# B&R Automation Studio project AAU12Segmenter (part 4)

### Config_1.assembly6d - X20CP1685/mapp6D/Config_1.assembly6d
```
Element gAssembly6D_1 (Type=assembly6d)
  Simulation6D = SimOff
  Shuttles:
    MaxShuttleCount = 8
    ShuttleIDMode = RealTimeID
    DefaultPosition:
      DefZ = 1.0
      DefRx = 0
      DefRy = 0
      DefRz = 0
    Limits:
      InPlaneLimits:
        InPlaneVelLim = 2
        InPlaneAccLim = 10
        InPlaneEmergDec = 1
      ShortAxLim:
        ShortAxAccLim:
          AccZLim = 10.0
          AccRxLim = 10.0
          AccRyLim = 10.0
          AccRzLim = 10.0
        ShortAxVelLim:
          VelZLim = 0.15
          VelRxLim = 0.1
          VelRyLim = 0.1
          VelRzLim = 0.3
  CyclicChannel6D:
    ReadChannel:
      Xaxis = TRUE
      Yaxis = TRUE
      Zaxis = TRUE
      Rxaxis = TRUE
      Ryaxis = TRUE
      Rzaxis = TRUE
  Fieldbus6D:
    SyncMode6D = ExternalPlkSync
    NodeNumber = 20
  IOMapp:
    Input = ::FBin
    Output = ::FBout
  Layout:
    Layout6D[1] = Layout6D_1
```

### Config_2.layout6d - X20CP1685/mapp6D/Config_2.layout6d
```
Element Layout6D_1 (Type=layout6d)
  Segments:
    SegRow = 4
    SegCol = 3
    Segment[1]:
      X = 0
      Y = 0
      Name
      IsMaster = True
    Segment[2]:
      X = 0
      Y = 1
      Name
      IsMaster = False
    Segment[3]:
      X = 0
      Y = 2
      Name
      IsMaster = False
    Segment[4]:
      X = 0
      Y = 3
      Name
      IsMaster = False
    Segment[5]:
      X = 1
      Y = 0
      Name
      IsMaster = False
    Segment[6]:
      X = 1
      Y = 1
      Name
      IsMaster = False
    Segment[7]:
      X = 1
      Y = 2
      Name
      IsMaster = False
    Segment[8]:
      X = 1
      Y = 3
      Name
      IsMaster = False
    Segment[9]:
      X = 2
      Y = 0
      Name
      IsMaster = False
    Segment[10]:
      X = 2
      Y = 1
      Name
      IsMaster = False
    Segment[11]:
      X = 2
      Y = 2
      Name
      IsMaster = False
    Segment[12]:
      X = 2
      Y = 3
      Name
      IsMaster = False
```

## Logical view

Binary libraries used (declarations not repeated): operator, runtime, astime, AsIecCon, standard, brdkSTR, AsSem, sys_lib, brsystem, AsBrStr, AsZip, FileIO, AsARCfg, AsEPL, AsIO, IecCheck, brdkViBase, brdkViCal, brdkViGeom, brdkViImg, brdkViMapp, brdkViVF, BRSE_RTK, AsHttp, powerlnk, MTLinAlg, ViBase 5.19.1, CoTrace 5.19.0, McBase, SfDomain 5.19.0, MpBase 5.19.0, McAcp6D, KUKAmxA3_1 3.01.1, AsUDP, asstring, KUKAmxA3_2 3.02.0, KUKAmxA3_3 3.03.1, KUKAmxA3_0 3.00.2

### Global.var - Global variables
```iecst
VAR
	FBin : Mc6DControllerFBIOType;
	FBout : Mc6DControllerFBIOType;
	GripperBlackPin : BOOL;
END_VAR
```

### Package Logical/Libraries - Global libraries

### Library Logical/Libraries/brdkMU (ANSIC) - BRDK machine unit library. Provides functionality to control machines.

#### brdkCM.typ
```iecst
TYPE
	brdk_cm_setup_typ : 	STRUCT  (*Equipment module setup structure.*)
		name : STRING[BRDK_MU_NAME_STRING_SIZE]; (*Name of the module.*)
		nameIdx : DINT := -1; (*Index to be added to name. If -1 no index will be set.*)
		parent : brdk_mu_setup_module_typ; (*Parameters to setup a parent module.*)
		sibling : ARRAY[0..BRDK_MU_MAX_SIBLINGS]OF brdk_mu_setup_module_typ; (*Enables the logging of the last state and sub state.*)
		status : brdk_cm_setup_status_typ; (*Enables the logging of the last state and sub state.*)
	END_STRUCT;
	brdk_cm_setup_status_typ : 	STRUCT  (*Enable or disable status functionality.*)
		state : BOOL := TRUE; (*State string.*)
		last : BOOL := TRUE; (*Last log entries.*)
	END_STRUCT;
	brdk_cm_status_typ : 	STRUCT  (*Control module status type.*)
		ready : BOOL := FALSE; (*Control module is ready for use.*)
		state : STRING[BRDK_MU_MAX_DESCRIPTION_STRING]; (*Can be set in the task to descripe what the module is doing in this state.*)
		time : UDINT; (*[ms] Actual time spend in the current state.*)
		last : ARRAY[0..BRDK_MU_MAX_LAST_SIZE]OF STRING[25]; (*The last state the module was in.*)
		cycleTime : UDINT; (*[µsec] Cycle time of the modules's task.*)
		parent : brdk_mu_status_module_typ; (*Information about the parent.*)
		sibling : ARRAY[0..BRDK_MU_MAX_SIBLINGS]OF brdk_mu_status_module_typ; (*List of available siblings.*)
		sleeping : BOOL; (*Indicates that the module is sleeping meaning that the module is not being executed because a new instance is being transferred.*)
		level : UDINT; (*Level in the hierarchy. Parent is level 0.*)
		name : STRING[BRDK_MU_NAME_STRING_SIZE]; (*Name of the module.*)
	END_STRUCT;
	brdk_cm_internal_mu_list_typ : 	STRUCT  (*Holds index's in the MU list.*)
		idx : DINT := -1; (*Own index in the mu list.*)
		parentIdx : DINT := -1; (*Parent index in the mu list.*)
		siblingIdx : ARRAY[0..BRDK_MU_MAX_SIBLINGS]OF DINT := [4(-1)]; (*Siblings index in the mu list.*)
	END_STRUCT;
	brdk_cm_internal_typ : 	STRUCT  (*Control module internal variables.*)
		initSubstate : UINT := 0; (*Internal temp sub state to be used in INIT PROGRAM.*)
		muList : brdk_cm_internal_mu_list_typ; (*Holds index's in the MU list.*)
		old : brdk_cm_state_old_typ; (*Holds the old states.*)
	END_STRUCT;
	brdk_cm_state_old_typ : 	STRUCT  (*Holds the old states.*)
		state : UINT; (*Old CM state.*)
		substate : UINT; (*Old CM substate.*)
	END_STRUCT;
END_TYPE
```

#### brdkEM.typ
```iecst
TYPE
	brdk_em_states_typ :
		( (*Module states. Based on ISA–TR88.00.02 state model.*)
		STATE_DEACTIVATED := 0, (*State Type: Wait
The module has not been activated yet. An activate command will cause an exit from
DEACTIVATED to a ACTIVATING state.*)
		STATE_CLEARING := 1, (*State Type: Acting
Initiated by a state command to clear faults that may have occurred
when ABORTING, and are present in the ABORTED state before
proceeding to a STOPPED state.*)
		STATE_STOPPED := 2, (*State Type: Wait
The machine is powered and stationary after completing the
STOPPING state. All communications with other systems are
functioning (if applicable). A Reset command will cause an exit from
STOPPED to the RESETTING state.*)
		STATE_STARTING := 3, (*State Type: Acting
This state provides the steps needed to start the machine and is a
result of a starting type command (local or remote). Following this
command the machine will begin to Execute.*)
		STATE_IDLE := 4, (*State Type: Wait
This is a state which indicates that RESETTING is complete. This
state maintains the machine conditions which were achieved during
the RESETTING state, and performs operations required when the
machine is in IDLE.*)
		STATE_SUSPENDED := 5, (*State Type: Wait
The machine may be running at a relevant set point speed, but
there is no product being produced while the machine is waiting for
external process conditions to return to normal. When the offending
process conditions return to normal, the SUSPENDED state will
transition to UNSUSPENDING and hence continue towards the
normal EXECUTE state.*)
		STATE_EXECUTE := 6, (*State Type: Dual
Once the machine is processing materials it is deemed to be
executing or in the EXECUTE state. Different machine modes will
result in specific types of EXECUTE activities. For example, if the
machine is in the Production mode, the EXECUTE will result in
products being produced, while in Clean Out mode the EXECUTE
state refers to the action of cleaning the machine.*)
		STATE_STOPPING := 7, (*State Type: Acting
This state executes the logic which brings the machine to a
controlled stop as reflected by the STOPPED state. Normal
STARTING of the machine can not be initiated unless RESETTING
had taken place.*)
		STATE_ABORTING := 8, (*State Type: Acting
The ABORTED state can be entered at any time in response to the
Abort command or on the occurrence of a machine fault. The
aborting logic will bring the machine to a rapid safe stop. Operation
of the emergency stop will cause the machine to be tripped by its
safety system. It will also provide a signal to initiate the
ABORTING State.*)
		STATE_ABORTED := 9, (*State Type: Wait
This state maintains machine status information relevant to the
Abort condition. The machine can only exit the ABORTED state
after an explicit Clear command, subsequently to manual
intervention to correct and reset the detected machine faults.*)
		STATE_HOLDING := 10, (*State Type: Acting
When the machine is in the EXECUTE state, the Hold command
can be used to start HOLDING logic which brings the machine to a
controlled stop or to a state which represents HELD for the
particular unit control mode. A machine can go into this state either
when an internal equipment fault is automatically detected or by an
operator command. The Hold command offers the operator a safe
way to intervene manually in the process (such as removing a
broken bottle from the in-feed) and restarting execution when
conditions are safe. To be able to restart production correctly after
the HELD state, all relevant process set-points and return status of
the procedures at the time of receiving the Hold command must be
saved in the machine controller when executing the HOLDING
procedure.*)
		STATE_HELD := 11, (*State Type: Wait
The HELD state holds the machine's operation while material
blockages are cleared, or to stop throughput while a downstream
problem is resolved, or enable the safe correction of an equipment
fault before the production may be resumed.*)
		STATE_UNHOLDING := 12, (*State Type: Acting
The UNHOLDING state is a response to an Operator command to
resume the EXECUTE state. Issuing the Unhold command will
retrieve the saved set-points and return the status conditions to
prepare the machine to re-enter the normal EXECUTE state.*)
		STATE_SUSPENDING := 13, (*State Type: Acting
This state is a result of a change in monitored conditions due to
process conditions or factors. The trigger event will cause a
temporary suspension of the EXECUTE state. SUSPENDING is
typically the result of starvation of upstream material in-feeds (i.e.,
container feed, beverage feed, crown feed, lubricant feed, etc.) that
is outside the dynamic speed control range or a downstream outfeed
blockage that prevents the machine from EXECUTING
continued steady production. During the controlled sequence of
SUSPENDING the machine will transition to a SUSPENDED state.
The SUSPENDING state might be forced by the operator.*)
		STATE_UNSUSPENDING := 14, (*State Type: Acting
This state is a result of a machine generated request from
SUSPENDED state to go back to the EXECUTE state. The actions
of this state may include ramping up speeds, turning on vacuums,
and the re-engagement of clutches. This state is done prior to
EXECUTE state, and prepares the machine for the EXECUTE state.*)
		STATE_RESETTING := 15, (*State Type: Acting
This state is the result of a RESET command from the STOPPED or
complete state. RESETTING will typically cause a machine to
sound a horn and place the machine in a state where components
are energized awaiting a START command.*)
		STATE_COMPLETING := 16, (*State Type: Acting
This state is an automatic response from the EXECUTE state.
Normal operation has run to completion (i.e., processing of material
at the infeed will stop).*)
		STATE_COMPLETE := 17, (*State Type: Wait
The machine has finished the COMPLETING state and is now
waiting for a Reset command before transitioning to the
RESETTING state.*)
		STATE_DEACTIVATING := 18, (*State Type: Acting
This state is the result of a disabled ACTIVATE command.*)
		STATE_ACTIVATING := 19 (*State Type: Acting
State between DEACTIVATED and STOPPED. This state is done prior to
STOPPED state, and prepares the machine for the STOPPED state.*)
		) := STATE_DEACTIVATED;
	brdk_em_activation_typ :
		( (*Type of activation of equipment module.*)
		BRDK_EM_ACTIVATE := 0, (*Activates the equipment module.*)
		BRDK_EM_DEACTIVATE := 1, (*Deactivated the equipment module.*)
		BRDK_EM_ACTIVATE_BY_PARENT := 2 (*Automatically follows it's parent activation.*)
		) := BRDK_EM_DEACTIVATE;
	brdk_em_command_typ : 	STRUCT  (*Equipment module commands. Based on ISATR88.00.02.*)
		abort : BOOL := FALSE; (*Abort --> Go to STATE_ABORTING - Can be set in all states.*)
		clear : BOOL := FALSE; (*Clear --> Go to STATE_STOPPING - Can only be set in STATE_ABORTED.*)
		stop : BOOL := FALSE; (*Stop --> Go to STATE_STOPPING - Can be set in all states.*)
		reset : BOOL := FALSE; (*Reset --> Go to STATE_RESETTING - Can only be set in STATE_STOPPED.*)
		start : BOOL := FALSE; (*Start --> Go to STATE_STARTING - Can only be set in STATE_IDLE, STATE_SUSPENDED, STATE_HELD.*)
		hold : BOOL := FALSE; (*Hold --> Go to STATE_HOLDING - Can only be set in STATE_EXECUTE.*)
		suspend : BOOL := FALSE; (*Suspend --> Go to STATE_SUSPENDING - Can only be set in STATE_EXECUTE.*)
		complete : BOOL := FALSE; (*Complete --> Go to STATE_COMPLETING - Can only be set in STATE_EXECUTE.*)
		sc : BOOL := FALSE; (*The State Complete indication within the Acting state procedure will cause a state transition to occur. Same functionality as subsuate = SC.*)
	END_STRUCT;
	brdk_em_setup_typ : 	STRUCT  (*Equipment module setup structure.*)
		name : STRING[BRDK_MU_NAME_STRING_SIZE]; (*Name of the module. If empty the name of the task will be given.*)
		nameIdx : DINT := -1; (*Index to be added to name. If -1 no index will be set.*)
		reactTo : brdk_em_setup_react_typ := BRDK_EM_REACT_TO_ALL; (*Indicates which parent state the module should react to.*)
		parent : brdk_mu_setup_module_typ; (*Parameters to setup a parent module.*)
		skipStopSC : BOOL := FALSE; (*When this parameter is set the module will stop even though is not in sub state SC.*)
		sibling : ARRAY[0..BRDK_MU_MAX_SIBLINGS]OF brdk_mu_setup_module_typ; (*List of siblings to a module.*)
		activation : brdk_em_activation_typ := BRDK_EM_ACTIVATE; (*Type of activation of equipment module.*)
		useSubstateSC : BOOL := FALSE; (*Enables the if substate is set to SC it will work as cmd.sc.*)
		restore : brdk_em_setup_restore_typ; (*Functionality to restore a module to it's state after a e.g. power failure.*)
		status : brdk_em_setup_status_typ; (*Enable or disable status functionality.*)
		customModeNames : ARRAY[0..BRDK_EM_MAX_CUSTOM_MODES]OF brdk_em_setup_custom_modes_typ; (*Custom mode names.*)
	END_STRUCT;
	brdk_em_setup_custom_modes_typ : 	STRUCT  (*Custom mode names.*)
		mode : DINT := 0; (*Mode integer value.*)
		modeName : STRING[BRDK_EM_MAX_MODE_NAME_SIZE] := ''; (*Mode name.*)
	END_STRUCT;
	brdk_em_setup_status_typ : 	STRUCT  (*Enable or disable status functionality.*)
		stateSubstateMode : BOOL := TRUE; (*State, sub state and mode strings.*)
		last : BOOL := TRUE; (*Last log entries.*)
		waitingFor : BOOL := TRUE; (*Waiting for.*)
		interruptedBy : BOOL := TRUE; (*interrupted by.*)
	END_STRUCT;
	brdk_em_setup_react_typ :
		( (*Indicates witch command/state the module should react to.*)
		BRDK_EM_REACT_TO_ALL := 0, (*Reacts to all states.*)
		BRDK_EM_REACT_TO_ABORT_AND_STOP := 1, (*Reacts only to abort and stop states.*)
		BRDK_EM_REACT_TO_ABORT_ONLY := 2, (*Reacts only to abort state.*)
		BRDK_EM_REACT_TO_STOP_ONLY := 3, (*Reacts only to stop state.*)
		BRDK_EM_REACT_TO_NONE := 4, (*Doesn't react to any state or mode change. Runs total independent. Equal to the old cmd.ignore.*)
		BRDK_EM_LISTEN_TO_ABORT_AND_STOP := 5, (*The module listen to it's parent aborting and stopping only. Parent don't react to the module.*)
		BRDK_EM_LISTEN_TO_ABORT_ONLY := 6, (*The module listen to it's parent aborting only. Parent don't react to the module.*)
		BRDK_EM_LISTEN_TO_STOP_ONLY := 7 (*The module listen to it's parent stopping only. Parent don't react to the module.*)
		) := BRDK_EM_REACT_TO_ALL;
	brdk_em_setup_restore_typ : 	STRUCT  (*Functionality to restore a module to it's state after a e.g. power failure.*)
		pRestoreStruct : REFERENCE TO brdk_em_restore_module_typ; (*Pointer to the restore structure. Must be defined directly in the task in order to make it retain/permanent.*)
		activate : BOOL := FALSE; (*Activates the storing of the module information in the restore structure. This is to avoid overwriting the restore information.*)
	END_STRUCT;
	brdk_em_status_typ : 	STRUCT  (*Equipment module status.*)
		state : STRING[21]; (*String representation of the state.*)
		substate : STRING[BRDK_MU_MAX_DESCRIPTION_STRING]; (*Can be set in the task to descripe what the module is doing in this substate.*)
		mode : STRING[21]; (*String representation of the mode.*)
		name : STRING[BRDK_MU_NAME_STRING_SIZE]; (*Name of the module. If empty the name of the task will be given.*)
		time : UDINT; (*[ms] Actual time spend in the current state.*)
		last : ARRAY[0..BRDK_MU_MAX_LAST_SIZE]OF STRING[43]; (*The last state and substate the module was in and the spend time.*)
		childCount : UDINT; (*How many children are registered.*)
		waitingFor : brdk_em_waiting_for_typ; (*Info: Which child the parent and the underlying modules are waiting for.*)
		interruptedBy : brdk_em_interrupted_by_typ; (*Info: Which child interruped the parent by going into STOPPING or ABORTING.*)
		color : brdk_em_color_typ; (*Color depending af the unit state.*)
		lightTree : brdk_em_status_light_tree_typ; (*Light tree indicating the status of the module.*)
		cycleTime : UDINT; (*[µsec] Cycle time of the modules's task.*)
		parent : brdk_mu_status_module_typ; (*Information about the parent.*)
		sibling : ARRAY[0..BRDK_MU_MAX_SIBLINGS]OF brdk_mu_status_module_typ; (*List of available siblings.*)
		unvalidatedCmd : BOOL; (*Indicates that the current state cannot accept the given command.*)
		unvalidatedMode : BOOL; (*Indicates that the current state cannot accept the given mode change. Modes can only be changed in STATE_STOPPED and in STATE_ACTIVATING. The status flag will be reset by a state change.*)
		sleeping : BOOL; (*Indicates that the module is sleeping meaning that the module is not being executed because a new instance is being transferred.*)
		level : UDINT; (*Level in the hierarchy. Parent is level 0.*)
	END_STRUCT;
	brdk_em_status_light_tree_typ : 	STRUCT  (*Light tree indicating the status of the module. The idea of the light tree status is that it can be mapped directly to an output module.*)
		red : BOOL := FALSE; (*Color red.*)
		yellow : BOOL := FALSE; (*Color yellow.*)
		blue : BOOL := FALSE; (*Color blue.*)
		green : BOOL := FALSE; (*Color green.*)
	END_STRUCT;
	brdk_em_color_typ :
		( (*Color to display the current state.*)
		GREY := 0, (*Wait State - Unit is disabled*)
		BLUE := 1, (*Wait State – A stable state used to identify that a Unit has achieved a defined set of
conditions. In such a state the Unit is holding or maintaining a status until transitioning
to an Acting state (White color). The unit is powered and stationary.*)
		WHITE := 2, (*Acting State – A state which represents some processing activity, for example ramping
up speed.
It implies the single or repeated execution of processing steps in a logical order, for a
finite time or until a specific condition has been reached, for example within the
Starting state the quality of the received data is checking, before raping up speed for
execution.*)
		GREEN := 3, (*Dual State - The Unit is in a stable acting state. The unit is running and drives are active
and the unit is producing.*)
		RED := 4, (*Wait state – A state which represents an error state on the Unit. In this state the Unit is
not producing, until the operator have managed to make a transition to the EXECUTING
state. The state holds the units operation in a safe environment, until the command
unhold are executed. For example a material blockage will move the unit into the HELD
state. The unit will leave the state HELD, when the operator have entered the unit,
removed the the bloackage, and enabled all safeguards and activated the Unhold
command.*)
		ORANGE := 5 (*Wait State – A state which represents an error state on the line and the Unit is running
at a relevant set point speed, but there is no product being produced while the unit is
waiting for external process conditions to return to normal. The unit will also enter this
state if the operator want to have a break.*)
		) := GREY;
	brdk_em_interrupted_by_typ : 	STRUCT  (*Tells which unit has interrupted the hierarchy into STATE_ABORTING or STATE_STOPPING.*)
		name : STRING[BRDK_MU_NAME_STRING_SIZE]; (*Name of the child that has interrupted the parent.*)
		state : brdk_em_states_typ := STATE_DEACTIVATED; (*State info.*)
		substate : UINT := 0; (*Substate info.*)
	END_STRUCT;
	brdk_em_waiting_for_typ : 	STRUCT  (*Tells which child module the hierarchy are waiting for. Can be that the modules are waiting for more children, but only one of them a shown at a time.*)
		name : STRING[BRDK_MU_NAME_STRING_SIZE]; (*Name of the child that the parent is waiting for.*)
		substate : STRING[BRDK_MU_MAX_DESCRIPTION_STRING]; (*Child substate.*)
	END_STRUCT;
	brdk_em_internal_typ : 	STRUCT  (*Internal variables.*)
		SemCreate_0 : SemCreate; (*Module semaphore.*)
		old : brdk_em_state_old_typ; (*Last state info.*)
		flashTime : UDINT := 0; (*Flash time counter.*)
		initSubstate : UINT := 0; (*Internal temp sub state to be used in STATE_DEACTIVATED.*)
		pInterrupter : UDINT := 0; (*Pointer to the module that interrupted.*)
		findParent : BOOL := FALSE; (*The module automatically finds it's parent's state.*)
		muList : brdk_em_internal_mu_list_typ; (*Holds index's in the MU list.*)
		cmdSC : BOOL; (*Internal command state complete.*)
		statusCnt : brdk_em_internal_status_cnt_typ; (*Status counter to indicate if a status change has been made.*)
		waitingForIdx : DINT := -1; (*Index of the module we are waiting for.*)
		deactivateRequest : BOOL := TRUE; (*A request to deactivate the mdule has been made.*)
		timeReminder : UDINT; (*Reminder of time when cycle time is below 1ms.*)
	END_STRUCT;
	brdk_em_internal_status_cnt_typ : 	STRUCT  (*Status counter to indicate if a status change has been made.*)
		internalCounter : DINT := -1; (*Internal counter which will be incremented if the status changes.*)
		externalCounter : DINT := -1; (*External counter which will hold the status counter of the waiting for module.*)
	END_STRUCT;
	brdk_em_state_old_typ : 	STRUCT  (*Holds the old states.*)
		state : brdk_em_states_typ := STATE_DEACTIVATED; (*Old state.*)
		substate : UINT := 0; (*Old substate.*)
		mode : DINT := 0; (*Old mode.*)
		reactTo : brdk_em_setup_react_typ := BRDK_EM_REACT_TO_ALL; (*Old reactTo.*)
	END_STRUCT;
	brdk_em_internal_mu_list_typ : 	STRUCT  (*Holds index's in the MU list.*)
		idx : DINT := -1; (*Own index in the mu list.*)
		parentIdx : DINT := -1; (*Parent index in the mu list.*)
		siblingIdx : ARRAY[0..BRDK_MU_MAX_SIBLINGS]OF DINT := [4(-1)]; (*Siblings index in the mu list.*)
		childrenIdx : ARRAY[0..BRDK_EM_MAX_CHILDREN]OF DINT; (*Children index in the mu list.*)
	END_STRUCT;
	brdk_em_restore_module_typ : 	STRUCT  (*Hold information that can be used to restore to it's active state in the case of a power failure.*)
		state : brdk_em_states_typ; (*Restored state.*)
		substate : UINT; (*Restored sub state.*)
		sc : BOOL; (*Restores state complete.*)
		mode : UINT; (*Restore mode.*)
	END_STRUCT;
	brdk_em_static_status_text_typ :
		( (*Internal enum to set a static status text*)
		STATUS_TEXT_DESCRIPTION := 0,
		STATUS_TEXT_ACTIVATION := 1
		);
END_TYPE
```

#### brdkMU.typ
```iecst
TYPE
	brdk_mu_setup_module_typ : 	STRUCT  (*Parameters to setup a connection to a module.*)
		name : STRING[BRDK_MU_NAME_STRING_SIZE]; (*Logical name of the module.*)
		index : DINT := -1; (*Index to be added to the module name. If -1 no index will be set.*)
	END_STRUCT;
	brdk_mu_status_module_typ : 	STRUCT  (*Status of a module.*)
		state : brdk_em_states_typ := STATE_DEACTIVATED; (*Module states. Based on ISA-TR88.00.02 state model.*)
		substate : UINT := 0; (*Equipment module substate can be used in the task. When a state is done set cmd.sc = true and the fb will take the unit to it's next state.*)
		sleeping : BOOL := FALSE; (*Indicates that the module is sleeping meaning that the module is not being executed because a new instance is being transferred.*)
		mode : DINT; (*Mode of the module.*)
		sc : BOOL; (*The State Complete indication within the Acting state procedure will cause a state transition to occur.*)
	END_STRUCT;
END_TYPE
```

#### brdkMU.fun
```iecst
FUNCTION_BLOCK brdkEM (*Represents an equipment module.*) (*$GROUP=User*)
	VAR_INPUT
		description : STRING[BRDK_MU_MAX_DESCRIPTION_STRING]; (*Description of what the substate is doing or waiting for.*)
		mode : DINT := MODE_PRODUCING; (*Control modes. Based on ISA-TR88.00.02 control modes. Modes can only be changed in STATE_STOPPED.*)
		cmd : brdk_em_command_typ; (*Control commands. Based on ISA-TR88.00.02 commands.*)
		setup : brdk_em_setup_typ; (*Setup of module.*)
		substate : UINT := 0; (*Equipment module substate can be used in the task. When a state is done set cmd.sc = true and the fb will take the unit to it's next state.*)
	END_VAR
	VAR_OUTPUT
		state : brdk_em_states_typ := STATE_DEACTIVATED; (*Equipment module state. State changes are controlled in the fb and is not allowed outside this fb. Based on ISA-TR88.00.02 states.*)
		status : brdk_em_status_typ; (*Module status.*)
	END_VAR
	VAR
		internal : brdk_em_internal_typ; (*Internal variables.*)
	END_VAR
END_FUNCTION_BLOCK

FUNCTION brdkEMSleep : DINT (*Put an equipment module to sleep. $RETURN=index;Index in the list.*) (*$GROUP=User,$CAT=User,$GROUPICON=User.png,$CATICON=User.png*)
	VAR_INPUT
		pEM : UDINT; (*Pointer to the equipment module.*)
	END_VAR
END_FUNCTION

FUNCTION brdkEMModeToA : UDINT (*Converts an equipment module mode int to a string representation. $RETURN=pointer;String pointer to mode string.*) (*$GROUP=User,$CAT=User,$GROUPICON=User.png,$CATICON=User.png*)
	VAR_INPUT
		mode : DINT := 0; (*Equipment module mode.*)
		pEM : UDINT := 0; (*Pointer to equipment module.*)
	END_VAR
END_FUNCTION

FUNCTION brdkEMStateToA : UDINT (*Converts an equipment module state enum to a string representation. $RETURN=pointer;String pointer to state string.*) (*$GROUP=User,$CAT=User,$GROUPICON=User.png,$CATICON=User.png*)
	VAR_INPUT
		state : brdk_em_states_typ; (*Equipment module state.*)
	END_VAR
END_FUNCTION

FUNCTION_BLOCK brdkCM (*Represents a control module. The module does not follow the ISA-TR88.00.02 standard.*) (*$GROUP=User,$CAT=User,$GROUPICON=User.png,$CATICON=User.png*)
	VAR_INPUT
		description : STRING[BRDK_MU_MAX_DESCRIPTION_STRING]; (*Description of what the state / substate is doing or waiting for.*)
		state : UINT := 0; (*Control module state must be used in the task.*)
		substate : UINT := 0; (*Control module substate must be used in the task.*)
		setup : brdk_cm_setup_typ; (*Setup of module.*)
	END_VAR
	VAR_OUTPUT
		status : brdk_cm_status_typ; (*Module status.*)
	END_VAR
	VAR
		internal : brdk_cm_internal_typ; (*Internal variables.*)
	END_VAR
END_FUNCTION_BLOCK

FUNCTION brdkCMSleep : DINT (*Put a control module to sleep. $RETURN=index;Index in the list.*) (*$GROUP=User,$CAT=User,$GROUPICON=User.png,$CATICON=User.png*)
	VAR_INPUT
		pCM : UDINT; (*Pointer to the control module.*)
	END_VAR
END_FUNCTION

FUNCTION brdkCMChangeParent : DINT (*Changes the parent of a control module. $RETURN=index;Index in the new parent.*) (*$GROUP=User,$CAT=User,$GROUPICON=User.png,$CATICON=User.png*)
	VAR_INPUT
		pCM : UDINT; (*Pointer to the control module.*)
		pParentName : UDINT; (*Pointert to the logical name of the parent module.*)
		parentIndex : DINT; (*Index to be added to the module name. If -1 no index will be set.*)
	END_VAR
END_FUNCTION

FUNCTION_BLOCK brdkUM (*Unit Machine / Information Receiver module. It makes communication with a remote system easy. This fb makes it possible to remote control an equipment module.*) (*$GROUP=User,$CAT=User,$GROUPICON=User.png,$CATICON=User.png*)
	VAR_INPUT
		mode : brdk_um_mode_typ := BRDK_UM_MODE_MANUAL; (*Communication mode.*)
		pEM : UDINT; (*Pointer to the main equipment module (machine unit).*)
		Status : brdk_um_pml_s_typ; (*Status tags.*)
		Admin : brdk_um_pml_a_typ; (*Administration tags.*)
	END_VAR
	VAR_OUTPUT
		Command : brdk_um_pml_c_typ; (*Command tags.*)
	END_VAR
	VAR
		internal : brdk_um_pml_internal_typ; (*Internal variables.*)
	END_VAR
END_FUNCTION_BLOCK
```

#### brdkMU_func.h
```c
#ifndef BRDK_MU_FUNCS
#define BRDK_MU_FUNCS 1

#include <brdkMU.h>
#include <bur/plctypes.h>

#ifdef __cplusplus
	extern "C"
	{
#endif

#ifdef __cplusplus
	};
#endif

#define false 0
#define true 1
#define NULL 0

extern SemCreate_typ SemCreateMUList;
extern unsigned char emListReady;

signed long addToMUList(unsigned long this, unsigned char type);
signed long getMUIndex(unsigned long this, brdk_mu_setup_module_typ* module);
brdkEM_typ* getEm(signed long idx);
signed long sleepMU(signed long idx, unsigned long this);
signed long wakeMU(signed long idx, unsigned long this);
unsigned long getCycleTime();
void updateSiblingInfo(signed long (*idxArr)[], brdk_mu_status_module_typ* status);
unsigned char moduleSleeping(signed long idx);

#endif /* !BRDK_MU_FUNCS */
```

#### brdkUM_func.h
```c
#ifndef BRDK_UM_FUNCS
#define BRDK_UM_FUNCS 1

#include <brdkMU_func.h>

void setCommand(signed long ctrlCmd, brdk_em_command_typ* emCmd, unsigned char value);
signed long cmdToState(signed long cmd);
void handleProductOverflow(brdk_um_pml_a_pc_typ* arr);

#endif /* !BRDK_UM_FUNCS */
```

#### brdkCM.c
```c
#include <brdkCM_func.h>

void brdkCM(struct brdkCM* this) {
	int i;
	brdkEM_typ* parent = getEm(this->internal.muList.parentIdx);
	brdk_mu_setup_module_typ module;

	/* initialize control module */
	switch(this->internal.initSubstate) {

		case 0:	/* this substate is only called in void _INIT / PROGRAM _INIT */
			if(this->setup.status.state) brdkStrCpy((unsigned long)this->status.state,(unsigned long)"initializing - looking for module pointers");
			if(this->setup.name[0] == 0) ST_name(0,(char*)&this->setup.name,(unsigned char)0); 														/* set module name to task name if not set*/
			brdkStrCpy((unsigned long)this->status.name,(unsigned long)this->setup.name);
			if(this->setup.nameIdx > -1) brdkStrAppendUdintToA(this->setup.nameIdx,(unsigned long)&this->status.name, BRDK_STR_CONVERT_DECIMAL,-1);	/* add index to task name */
			this->internal.muList.parentIdx = -1;
			for(i=0; i<= BRDK_MU_MAX_SIBLINGS; i++) this->internal.muList.siblingIdx[i] = -1;
			this->internal.initSubstate = 10;
			break;

		case 10:
			if(!emListReady) {
				if(this->setup.status.state) brdkStrCpy((unsigned long)this->status.state,(unsigned long)"waiting for mu list to be ready");
			}
			else {
				brdkStrCpy((unsigned long)module.name,(unsigned long)this->setup.name);
				module.index = this->setup.nameIdx;
				this->internal.muList.idx = getMUIndex((unsigned long)this, &module);
				if(this->internal.muList.idx != -1) {
					wakeMU(this->internal.muList.idx,(unsigned long)this);
					if(this->setup.status.last) {
						brdkStrMemMove((unsigned long)this->status.last[1],(unsigned long)this->status.last[0], sizeof(this->status.last[0])*BRDK_MU_MAX_LAST_SIZE);
						brdkStrCpy((unsigned long)this->status.last[0],(unsigned long)"module awake");
					}
					this->internal.initSubstate = 65001;
				}
				else {
					if(SemAcquire(SemCreateMUList.ident) != ERR_OK) {
						if(this->setup.status.state) brdkStrCpy((unsigned long)this->status.state,(unsigned long)"waiting global semaphore to be free");
					}
					else {
						this->internal.muList.idx = addToMUList((unsigned long)this,0);
						SemRelease(SemCreateMUList.ident);
						if(this->setup.status.state) brdkStrCpy((unsigned long)this->status.state,(unsigned long)"module added em list");
						if(this->internal.muList.idx != -1) this->internal.initSubstate = !this->setup.parent.name[0] ? 40 : 30;	/* check if the module has a parent name assigned */
						else {
							if(this->setup.status.state) brdkStrCpy((unsigned long)this->status.state,(unsigned long)"em list full. Expand BRDK_EM_MAX_EMS.");
							this->internal.initSubstate = 200;
						}
					}
				}
			}

		case 30:	/* find parent */
			this->internal.muList.parentIdx = getMUIndex((unsigned long)this, &this->setup.parent);
			if(this->internal.muList.parentIdx == -1) {
				if(this->setup.status.state) brdkStrCpy((unsigned long)this->status.state,(unsigned long)"parent not found");
			}
			else this->internal.initSubstate = 40;
			break;

		case 40:	/* find siblings */
			for(i=0; i<= BRDK_MU_MAX_SIBLINGS; i++) {
				if(this->setup.sibling[i].name[0] != 0) {
					this->internal.muList.siblingIdx[i] = getMUIndex((unsigned long)this, &this->setup.sibling[i]);
					if(this->internal.muList.siblingIdx[i] == -1) {
						if(this->setup.status.state) {
							brdkStrCpy((unsigned long)this->status.state,(unsigned long)"sibling: ");
							brdkStrCat((unsigned long)this->status.state,(unsigned long)this->setup.sibling[i].name);
							brdkStrCat((unsigned long)this->status.state,(unsigned long)" not found");
						}
						break;
					}
				}
			}
			if(i>=BRDK_MU_MAX_SIBLINGS) {
				this->status.state[0] = 0;	/* reset status text */
				this->internal.initSubstate = 65000;
			}
			break;

		case 65000:	/* module ready */
			/* check if status is not set */
			if(this->status.state[0] == 0 && this->setup.status.state) {
				brdkStrUdintToA(this->state,(unsigned long)this->status.state,BRDK_STR_CONVERT_DECIMAL);
				if(this->substate != 0) {
					brdkStrCat((unsigned long)this->status.state,(unsigned long)": ");
					brdkStrAppendUdintToA(this->substate,(unsigned long)this->status.state,BRDK_STR_CONVERT_DECIMAL,-1);
				}
				if(this->description[0] != 0) {
					brdkStrCat((unsigned long)this->status.state,(unsigned long)": ");
					brdkStrCat((unsigned long)this->status.state,(unsigned long)this->description);
				}
			}

			/* state change */
			if(this->state != this->internal.old.state || this->substate != this->internal.old.substate) {
				/* save last state for log */
				if(this->setup.status.last) {
					brdkStrMemMove((unsigned long)this->status.last[1],(unsigned long)this->status.last[0], sizeof(this->status.last[0])*BRDK_MU_MAX_LAST_SIZE);
					brdkStrUdintToA(this->internal.old.state,(unsigned long)this->status.last[0],BRDK_STR_CONVERT_DECIMAL);
					brdkStrCat((unsigned long)this->status.last[0],(unsigned long)": ");
					if(this->internal.old.substate || this->substate != 0) {	/* if the substate != 0 then we also want to log the oldsubstate even if it's 0 */
						brdkStrAppendUdintToA(this->internal.old.substate,(unsigned long)this->status.last[0],BRDK_STR_CONVERT_DECIMAL,-1);
						brdkStrCat((unsigned long)this->status.last[0], (unsigned long)": ");
					}
					brdkStrAppendUdintToA(this->status.time, (unsigned long)this->status.last[0],BRDK_STR_CONVERT_DECIMAL,-1);
					brdkStrCat((unsigned long)this->status.last[0], (unsigned long)"ms");
				}
				/* reset */
				if(this->state != this->internal.old.state) this->substate = 0;	/* if the state has been changed the substate will be reset */
				this->status.state[0] = this->description[0] = 0;
				this->internal.old.state = this->state;
				this->internal.old.substate = this->substate;
				this->status.time = 0;
			}
			else this->status.time += this->status.cycleTime/1000;

			/* update parent info */
			if(parent != NULL) {
				this->status.parent.state = parent->state;
				this->status.parent.substate = parent->substate;
				this->status.parent.sleeping = parent->status.sleeping;
				this->status.parent.sc = parent->cmd.sc;
			}

			/* update siblings info */
			updateSiblingInfo(&this->internal.muList.siblingIdx, &this->status.sibling[0]);

			this->status.level = parent != NULL ? parent->status.level+1 : 0;	/* sets the hierarchy level */

			break;

	}

	if(!this->status.cycleTime) this->status.cycleTime = getCycleTime();	/* get the modules cycle time */
	this->status.ready = this->internal.initSubstate == 65000;

}
```

#### brdkCMChangeParent.c
```c
#include <brdkMU_func.h>

signed long brdkCMChangeParent(unsigned long pCM, unsigned long pParentName, signed long parentIndex) {
	signed long tmpIdx = 0;
	brdk_mu_setup_module_typ module;
	brdkCM_typ* this;
	if(pCM != 0 && pParentName != 0 && emListReady) {
		this = (brdkCM_typ*)pCM;
		brdkStrCpy((unsigned long)module.name,pParentName);
		module.index = parentIndex;
		tmpIdx = getMUIndex((unsigned long)this, &module);
		if(tmpIdx != -1) {
			this->internal.muList.parentIdx = tmpIdx;
			brdkStrCpy((unsigned long)this->setup.parent.name,(unsigned long)module.name);
			this->setup.parent.index = module.index;
			return this->internal.muList.parentIdx;
		}
	}
	return -1;
}
```

#### brdkEM_func.c
```c
#include <brdkEM_func.h>

static unsigned char semCreator = false;
SemCreate_typ SemCreateMUList;
char tmpStr[BRDK_MU_MAX_DESCRIPTION_STRING];

/* initialize the equipment module */
void brdkEMInitialize(brdkEM_typ* this, brdkEM_typ* parent) {
	int i;
	brdk_mu_setup_module_typ module;

	switch(this->internal.initSubstate) {

		case 0:
			if(this->setup.name[0] == 0) ST_name(0,(char*)&this->setup.name,(unsigned char)0); 														/* set module name to task name if not set*/
			brdkStrCpy((unsigned long)this->status.name,(unsigned long)this->setup.name);
			if(this->setup.status.stateSubstateMode) {
				brdkStrCpy((unsigned long)this->status.state,(unsigned long)brdkEMStateToA(this->state));
				brdkStrCpy((unsigned long)this->status.mode,brdkEMModeToA(this->mode, this));
			}
			if(this->setup.nameIdx > -1) brdkStrAppendUdintToA(this->setup.nameIdx,(unsigned long)&this->status.name, BRDK_STR_CONVERT_DECIMAL,-1);	/* add index to task name */
			this->internal.muList.parentIdx = -1;
			for(i=0; i<= BRDK_EM_MAX_CHILDREN; i++) this->internal.muList.childrenIdx[i] = -1;
			for(i=0; i<= BRDK_MU_MAX_SIBLINGS; i++) this->internal.muList.siblingIdx[i] = -1;
			if(!semCreator) {
				setSubStateText(this,(unsigned long)"creating global semaphore");
				semCreator = true;
				this->internal.initSubstate = 10;
			}
			else this->internal.initSubstate = 20;
			break;

		case 10:
			SemCreateMUList.enable = true;
			SemCreateMUList.initCount = 0;
			SemCreateMUList.maxCount = 1;
			SemCreate(&SemCreateMUList);
			if(SemCreateMUList.status != ERR_OK) setSubStateText(this,(unsigned long)"creating global semaphore");
			else {
				SemRelease(SemCreateMUList.ident);
				this->internal.muList.idx = addToMUList((unsigned long)this,0);
				if(this->internal.muList.idx != -1) {
					emListReady = true;
					this->internal.initSubstate = !this->setup.parent.name[0] ? 40 : 30;	/* check if the module has a parent name assigned */
				}
				else {
					setSubStateText(this,(unsigned long)"em list full. Expand BRDK_EM_MAX_EMS.");
					this->internal.initSubstate = 200;
				}
			}
			break;

		case 20:	/* add module to em list */
			if(!emListReady) setSubStateText(this,(unsigned long)"waiting for em list to be ready");
			else {
				brdkStrCpy((unsigned long)module.name,(unsigned long)this->setup.name);
				module.index = this->setup.nameIdx;
				this->internal.muList.idx = getMUIndex((unsigned long)this, &module);
				if(this->internal.muList.idx != -1) {
					if(moduleSleeping(this->internal.muList.idx)) {
						wakeMU(this->internal.muList.idx,(unsigned long)this);
						if(this->setup.status.last) {
							brdkStrMemMove((unsigned long)this->status.last[1],(unsigned long)this->status.last[0], sizeof(this->status.last[0])*BRDK_MU_MAX_LAST_SIZE);
							brdkStrCpy((unsigned long)this->status.last[0],(unsigned long)"module awake");
						}
						this->internal.initSubstate = 65000;
					}
					else {	/* module name already exists in the list */
						this->status.substate[0] = 0;	/* reset sub state text */
						if(this->setup.status.stateSubstateMode) {
							brdkStrCpy((unsigned long)tmpStr,(unsigned long)"module name ");
							brdkStrCat((unsigned long)tmpStr,(unsigned long)module.name);
							brdkStrCat((unsigned long)tmpStr,(unsigned long)" already used. Rename module.");
							setSubStateText(this,(unsigned long)tmpStr);
						}
						this->internal.muList.idx = -1;
						this->internal.initSubstate = 100;
					}
				}
				else {
					if(SemAcquire(SemCreateMUList.ident) != ERR_OK) setSubStateText(this,(unsigned long)"waiting global semaphore to be free");
					else {
						this->internal.muList.idx = addToMUList((unsigned long)this,0);
						SemRelease(SemCreateMUList.ident);
						setSubStateText(this,(unsigned long)"module added em list");
						if(this->internal.muList.idx != -1) this->internal.initSubstate = !this->setup.parent.name[0] ? 40 : 30;	/* check if the module has a parent name assigned */
						else {
							setSubStateText(this,(unsigned long)"em list full. Expand BRDK_EM_MAX_EMS.");
							this->internal.initSubstate = 200;
						}
					}
				}
			}
			break;

		case 30:	/* find parent */
			this->internal.muList.parentIdx = getMUIndex((unsigned long)this, &this->setup.parent);
			if(this->internal.muList.parentIdx == -1) setSubStateText(this,(unsigned long)"parent not found");
			else this->internal.initSubstate = 40;
			break;

		case 40:	/* find siblings */
			for(i=0; i<= BRDK_MU_MAX_SIBLINGS; i++) {
				if(this->setup.sibling[i].name[0] != 0) {
					this->internal.muList.siblingIdx[i] = getMUIndex((unsigned long)this, &this->setup.sibling[i]);
					if(this->internal.muList.siblingIdx[i] == -1) {
						if(this->setup.status.stateSubstateMode) {
							brdkStrCpy((unsigned long)tmpStr,(unsigned long)"sibling: ");
							brdkStrCat((unsigned long)tmpStr,(unsigned long)this->setup.sibling[i].name);
							brdkStrCat((unsigned long)tmpStr,(unsigned long)" not found");
							setSubStateText(this,(unsigned long)tmpStr);
						}
						break;
					}
				}
			}
			if(i>=BRDK_MU_MAX_SIBLINGS) {
				this->status.substate[0] = 0;	/* reset status text */
				this->internal.initSubstate = this->internal.SemCreate_0.ident == 0 ? 50 : 60;
			}
			break;

		case 50:
			this->internal.SemCreate_0.enable = true;
			this->internal.SemCreate_0.initCount = 0;
			this->internal.SemCreate_0.maxCount = 1;
			SemCreate(&this->internal.SemCreate_0);
			switch(this->internal.SemCreate_0.status) {

				case 0:	/* ERR_OK */
					SemRelease(this->internal.SemCreate_0.ident);		/* release the semaphore so it's ready */
					this->internal.initSubstate = 60;
					break;

				case 65535:	/* ERR_FUB_BUSY */
					break;

				default:
					setSubStateText(this,(unsigned long)"error creating the semaphore");
					break;

			}
			break;

		case 60:
			switch(this->setup.activation) {
				case BRDK_EM_ACTIVATE:
					this->internal.deactivateRequest = false;
					this->internal.initSubstate = 70;
					break;

				case BRDK_EM_ACTIVATE_BY_PARENT:
					if(parent != NULL) {
						if(!parent->internal.deactivateRequest) {
							this->internal.initSubstate = 70;
							this->internal.deactivateRequest = false;
						}
					}
					break;

				default: break;

			}
			break;

		case 70:
			setSubStateText(this,(unsigned long)"register child to parent");
			if(RegisterChild(this, parent) == 0) {
				this->internal.initSubstate = 65000;				/* add child to parent's children list */
				if(this->substate == 0) this->substate = 65000;		/* if substate is still 0 it's auto set to SC */
			}
			break;

		case 100: /* error module name already used. Check if anme is being changed */
			break;

	}
}

/* traverse and find the real interrupter */
unsigned long findInterrupter(unsigned long pEM) {
	if(((brdkEM_typ*)pEM)->internal.pInterrupter != pEM) return findInterrupter(((brdkEM_typ*)pEM)->internal.pInterrupter);
	return pEM;
}

/* flash functionality */
brdk_em_color_typ flashColor(brdkEM_typ* this, brdk_em_color_typ color) {
	if(this->internal.flashTime >= BRDK_EM_FLASH_TIME*2) this->internal.flashTime = 0;
	else this->internal.flashTime += this->status.cycleTime/1000;
	return this->internal.flashTime >= BRDK_EM_FLASH_TIME ? color : WHITE;
}

/* light tree functionality */
void lightTree(brdkEM_typ* this, brdk_em_color_typ color1, brdk_em_color_typ color2) {
	this->status.lightTree.red 		= color1 == RED || color2 == RED;
	this->status.lightTree.yellow 	= color1 == ORANGE || color2 == ORANGE;
	this->status.lightTree.blue 	= color1 == BLUE || color2 == BLUE;
	this->status.lightTree.green 	= color1 == GREEN || color2 == GREEN;
}

/* set default sub state text if not set in program */
void setSubStateText(brdkEM_typ* this, unsigned long pStr) {
	const int MAX_COUNTER = 99999;
	if(this->status.substate[0] == 0 && this->setup.status.stateSubstateMode) {
		if(pStr != 0) {
			brdkStrCpy((unsigned long)this->status.substate,pStr);
			this->internal.statusCnt.internalCounter = this->internal.statusCnt.internalCounter > MAX_COUNTER ? 0 : this->internal.statusCnt.internalCounter+1;		/* increase the status counter to indicate that a change was made */
		}
		else {
			if(this->description[0] == 0) {
				if(this->substate == 0) {
					brdkStrCpy((unsigned long)this->status.substate,(unsigned long)"0: waiting for state change (SC)");
					this->internal.statusCnt.internalCounter = this->internal.statusCnt.internalCounter > MAX_COUNTER ? 0 : this->internal.statusCnt.internalCounter+1;		/* increase the status counter to indicate that a change was made */
				}
				else if(this->internal.cmdSC) {
					switch(this->state) {
						case STATE_DEACTIVATED: brdkStrCpy((unsigned long)this->status.substate, (unsigned long)"SC: waiting for activate command"); break;
						case STATE_STOPPED: case STATE_COMPLETE: brdkStrCpy((unsigned long)this->status.substate, (unsigned long)"SC: waiting for reset command"); break;
						case STATE_IDLE: case STATE_SUSPENDED: case STATE_HELD:	brdkStrCpy((unsigned long)this->status.substate, (unsigned long)"SC: waiting for start command"); break;
						case STATE_ABORTED: brdkStrCpy((unsigned long)this->status.substate, (unsigned long)"SC: waiting for clear command"); break;
						default: brdkStrCpy((unsigned long)this->status.substate, (unsigned long)"SC: waiting for command"); break;
					}
					this->internal.statusCnt.internalCounter = this->internal.statusCnt.internalCounter > MAX_COUNTER ? 0 : this->internal.statusCnt.internalCounter+1;		/* increase the status counter to indicate that a change was made */
				}
			}
			else {
				brdkStrUdintToA(this->substate,(unsigned long)&this->status.substate,BRDK_STR_CONVERT_DECIMAL);
				brdkStrCat((unsigned long)this->status.substate, (unsigned long)": ");
				brdkStrCat((unsigned long)this->status.substate, (unsigned long)this->description);
				this->internal.statusCnt.internalCounter = this->internal.statusCnt.internalCounter > MAX_COUNTER ? 0 : this->internal.statusCnt.internalCounter+1;		/* increase the status counter to indicate that a change was made */
			}
		}
	}
}

/* if the parent mode is changed we also changes it for alle the children */
void setChildrenMode(brdkEM_typ* this) {
	int i;
	for(i=0; i <= BRDK_EM_MAX_CHILDREN; i++) {
		brdkEM_typ* child = getEm(this->internal.muList.childrenIdx[i]);
		if(child != NULL) {
			if(this->setup.reactTo == BRDK_EM_REACT_TO_NONE) child->mode = child->mode;
			else child->mode = this->mode;
		}
		else break;
	}
}

/* CHECKS IF ALL THE CHILDREN IS IN STATE */
void checkChildren(brdkEM_typ* this, brdk_em_states_typ STATE) {
	brdkEM_typ* parent;
	brdkEM_typ* child;
	if(this->internal.cmdSC) {
		int i = 0, j;
		while(i < this->status.childCount) {
			child = getEm(this->internal.muList.childrenIdx[i]);
			if(child != NULL) {
				j = i;
				if(child->state == STATE_ACTIVATING || child->state == STATE_DEACTIVATED || child->state == STATE_DEACTIVATING) i++;
				else {
					switch(child->setup.reactTo) {

						case BRDK_EM_REACT_TO_ALL:
							if(child->state == STATE) i++;
							break;

						case BRDK_EM_REACT_TO_ABORT_AND_STOP:
							if(STATE == STATE_ABORTED || STATE == STATE_STOPPED) {
								if(child->state == STATE) i++;
							}
							else i++;
							break;

						case BRDK_EM_REACT_TO_ABORT_ONLY:
							if(STATE == STATE_ABORTED) {
								if(child->state == STATE) i++;
							}
							else i++;
							break;

						case BRDK_EM_REACT_TO_STOP_ONLY:
							if(STATE == STATE_STOPPED) {
								if(child->state == STATE) i++;
							}
							else i++;
							break;

						case BRDK_EM_REACT_TO_NONE: case BRDK_EM_LISTEN_TO_ABORT_AND_STOP: case BRDK_EM_LISTEN_TO_ABORT_ONLY: case BRDK_EM_LISTEN_TO_STOP_ONLY:
							i++;
							break;

					}
				}
				if(j == i) {	/* index not increased */
					if(child->internal.waitingForIdx != -1) {	/* check to see if a child is also waiting for someone */
						if(this->internal.waitingForIdx != child->internal.waitingForIdx) { /* check if the index has changed - otherwise there is nothing to update in the name */
							if(this->setup.status.waitingFor) brdkStrCpy((unsigned long)this->status.waitingFor.name,(unsigned long)child->status.waitingFor.name);
							this->internal.waitingForIdx = child->internal.waitingForIdx;
						}
						if(this->internal.statusCnt.externalCounter != child->internal.statusCnt.externalCounter) {	/* check if there is a change in the status text */
							if(this->setup.status.waitingFor) brdkStrCpy((unsigned long)this->status.waitingFor.substate,(unsigned long)child->status.waitingFor.substate);
							this->internal.statusCnt.externalCounter = child->internal.statusCnt.externalCounter;
						}
					}
					else {
						if(this->internal.waitingForIdx != child->internal.muList.idx) { /* check if the index has changed - otherwise there is nothing to update in the name */
							if(this->setup.status.stateSubstateMode) {
								brdkStrCpy((unsigned long)this->status.waitingFor.name,(unsigned long)child->setup.name);
								brdkStrCpy((unsigned long)tmpStr, (unsigned long)"SC: waiting for ");
								brdkStrCat((unsigned long)tmpStr, (unsigned long)this->status.waitingFor.name);
								setSubStateText(this,(unsigned long)tmpStr);
							}
							this->internal.waitingForIdx = child->internal.muList.idx;
						}
						if(this->internal.statusCnt.externalCounter != child->internal.statusCnt.internalCounter) {	/* check if there is a change in the status text */
							if(this->setup.status.waitingFor) brdkStrCpy((unsigned long)this->status.waitingFor.substate,(unsigned long)child->status.substate);
							this->internal.statusCnt.externalCounter = child->internal.statusCnt.internalCounter;
						}
					}
					break;
				}
			}
			else break;
		}
		if(parentStateOK(this)) {
			if(i==this->status.childCount) {
				if(this->state == STATE_RESETTING || this->state == STATE_CLEARING) {	/* clear interrupted by data */
					brdkStrMemSet((unsigned long)&this->status.interruptedBy,0,sizeof(this->status.interruptedBy));
					this->internal.pInterrupter = 0;
				}
				if(this->internal.waitingForIdx != -1) {
					if(this->setup.status.waitingFor) brdkStrMemSet((unsigned long)&this->status.waitingFor,0,sizeof(this->status.waitingFor)); /* clear waiting for data */
					this->internal.waitingForIdx = -1;				/* reset waiting for index */
					this->internal.statusCnt.externalCounter = -1;	/* reset external status counter */
				}
				this->state = STATE;
			}
		}
		else {
			if(!this->status.waitingFor.name[0]) {
				parent = getEm(this->internal.muList.parentIdx);
				if(parent != NULL) {
					if(this->internal.waitingForIdx != parent->internal.muList.idx) { /* check if the index has changed - otherwise there is nothing to update */
						this->internal.waitingForIdx = parent->internal.muList.idx;
						if(parent->state == STATE_DEACTIVATED || parent->state == STATE_DEACTIVATING) setSubStateText(this,(unsigned long)"SC: parent is deactivated");
						else setSubStateText(this,(unsigned long)"SC: waiting for parent");
						if(this->setup.status.waitingFor) brdkStrCpy((unsigned long)this->status.waitingFor.name,(unsigned long)parent->setup.name);
					}
					if(this->internal.statusCnt.externalCounter != parent->internal.statusCnt.internalCounter) {	/* check if there is a change in the status text */
						if(this->setup.status.waitingFor) brdkStrCpy((unsigned long)this->status.waitingFor.substate,(unsigned long)parent->status.substate);
						this->internal.statusCnt.externalCounter = parent->internal.statusCnt.internalCounter;
					}
				}
			}
		}
	}
}

/* make sure eventual parent is also in same state before state change */
int parentStateOK(brdkEM_typ* this) {
	int status = false;
	brdkEM_typ* parent = getEm(this->internal.muList.parentIdx);
	if(parent != NULL) {
		switch(this->setup.reactTo) {
			case BRDK_EM_REACT_TO_ALL: 				status = (parent->state == this->state || this->internal.findParent); break;
			case BRDK_EM_REACT_TO_ABORT_AND_STOP: 	status = (this->state == STATE_ABORTING || this->state == STATE_STOPPING) ? (parent->state == this->state) : true; break;
			case BRDK_EM_REACT_TO_ABORT_ONLY:		status = (this->state == STATE_ABORTING) ? (parent->state == this->state) : true; break;
			case BRDK_EM_REACT_TO_STOP_ONLY:		status = (this->state == STATE_STOPPING) ? (parent->state == this->state) : true; break;
			case BRDK_EM_REACT_TO_NONE: case BRDK_EM_LISTEN_TO_ABORT_AND_STOP: case BRDK_EM_LISTEN_TO_ABORT_ONLY: case BRDK_EM_LISTEN_TO_STOP_ONLY:	status = true;
		}
	}
	else status = true;
	return status;
}

/* automatically take the module to it's parents state */
void findParent(brdkEM_typ* this, brdkEM_typ* parent, brdk_em_states_typ cmd, int numArgs, ...) {
	if(parent != NULL) {
		va_list list;
		int i;
		if(this->state == parent->state) this->internal.findParent = false;
		else {
			va_start(list, numArgs);
			for(i=0; i < numArgs; i++) {
				brdk_em_states_typ checkState = va_arg(list, brdk_em_states_typ);
				if(parent->state == checkState) {
					switch(cmd) {
						case STATE_RESETTING: this->cmd.reset = true; break;
						case STATE_STARTING: case STATE_UNHOLDING: case STATE_UNSUSPENDING: this->cmd.start = true; break;
						case STATE_EXECUTE:
							switch(checkState) {
								case STATE_HOLDING: case STATE_HELD: this->cmd.hold = true; break;
								case STATE_SUSPENDING: case STATE_SUSPENDED: this->cmd.suspend = true; break;
								case STATE_COMPLETING: case STATE_COMPLETE: this->cmd.complete = true; break;
								default: break;
							}
							break;
						default: break;
					}
				}
			}
		}
	}
}

/* observes if one of the children is in one of the states */
void observeChildrensState(brdkEM_typ* this, int numArgs, ...) {
	int i,j;
	brdkEM_typ* child;
	va_list list;																					/* define argument list variable */
	for(i=0; i <= BRDK_EM_MAX_CHILDREN; i++) {														/* check all children */
		child = getEm(this->internal.muList.childrenIdx[i]);
		if(child != NULL) {											/* */
			brdk_em_setup_react_typ reactTo = child->setup.reactTo;
			if(reactTo == BRDK_EM_REACT_TO_NONE || reactTo == BRDK_EM_REACT_TO_NONE || reactTo == BRDK_EM_LISTEN_TO_ABORT_AND_STOP || reactTo == BRDK_EM_LISTEN_TO_ABORT_ONLY || reactTo == BRDK_EM_LISTEN_TO_STOP_ONLY) this->state = this->state;
			else {
				va_start(list, numArgs);
				for(j=0; j < numArgs; j++) {
					brdk_em_states_typ child_state = va_arg(list, brdk_em_states_typ);
					if(child->state == child_state) {
						switch(child_state) {

							case STATE_ABORTING:
								if(reactTo == BRDK_EM_REACT_TO_ALL || reactTo == BRDK_EM_REACT_TO_ABORT_AND_STOP || reactTo == BRDK_EM_REACT_TO_ABORT_ONLY) {
									this->internal.pInterrupter = findInterrupter((unsigned long)child); /* save who went in aborted or aborting */
									this->state = STATE_ABORTING;
								}
								break;

							case STATE_STOPPING:
								if((this->internal.cmdSC || this->setup.skipStopSC) && (reactTo == BRDK_EM_REACT_TO_ALL || reactTo == BRDK_EM_REACT_TO_ABORT_AND_STOP || reactTo == BRDK_EM_REACT_TO_STOP_ONLY)) {
									this->internal.pInterrupter = findInterrupter((unsigned long)child); /* save who went in stopped or stopping */
									this->state = STATE_STOPPING;
								}
								break;

							case STATE_SUSPENDING:
								if(this->internal.cmdSC && reactTo == BRDK_EM_REACT_TO_ALL) {
									this->internal.pInterrupter = findInterrupter((unsigned long)child); /* save who went in suspending or suspended */
									this->state = STATE_SUSPENDING;
								}
								break;

							case STATE_HOLDING:
								if(this->internal.cmdSC && reactTo == BRDK_EM_REACT_TO_ALL) {
									this->internal.pInterrupter = findInterrupter((unsigned long)child); /* save who went in holding or held */
									this->state = STATE_HOLDING;
								}
								break;

							default:
								break;

						}
						va_end(list);
						break;
					}
				}
			}
		}
		else {
			va_end(list);
			break;
		}
	}
}

/* observes the parent state by the given states */
void observeParentState(brdkEM_typ* this, brdkEM_typ* parent, int numArgs, ...) {
	int i;
	brdk_em_setup_react_typ reactTo =  this->setup.reactTo;
	if(parent == NULL || reactTo == BRDK_EM_REACT_TO_NONE) this->state = this->state;
	else {
		va_list list;																									/* define argument list variable */
		va_start(list, numArgs);																						/* init list */
		for(i=0; i < numArgs; i++) if(parent->state==va_arg(list, brdk_em_states_typ)) {
			switch(parent->state) {

				case STATE_ABORTING:
					if(reactTo == BRDK_EM_REACT_TO_ALL || reactTo == BRDK_EM_REACT_TO_ABORT_AND_STOP || reactTo == BRDK_EM_REACT_TO_ABORT_ONLY || reactTo == BRDK_EM_LISTEN_TO_ABORT_AND_STOP || reactTo == BRDK_EM_LISTEN_TO_ABORT_ONLY) {
						this->state = parent->state; 	/* get next state item and check if it's equal to parent state. and then set chils state*/
						this->internal.pInterrupter = parent->internal.pInterrupter;
					}
					break;

				case STATE_STOPPING:
					if((this->internal.cmdSC || this->setup.skipStopSC) && (reactTo == BRDK_EM_REACT_TO_ALL || reactTo == BRDK_EM_REACT_TO_ABORT_AND_STOP || reactTo == BRDK_EM_REACT_TO_STOP_ONLY || reactTo == BRDK_EM_LISTEN_TO_STOP_ONLY)) {
						this->state = parent->state; 	/* get next state item and check if it's equal to parent state. and then set chils state*/
						this->internal.pInterrupter = parent->internal.pInterrupter;
					}
					break;

				case STATE_CLEARING:
					if(this->internal.cmdSC && (reactTo == BRDK_EM_REACT_TO_ALL || reactTo == BRDK_EM_REACT_TO_ABORT_AND_STOP || reactTo == BRDK_EM_REACT_TO_ABORT_ONLY)) this->state = parent->state; 	/* get next state item and check if it's equal to parent state. and then set chils state*/
					break;

				default:
					if(this->internal.cmdSC && reactTo == BRDK_EM_REACT_TO_ALL) this->state = parent->state; 	/* get next state item and check if it's equal to parent state. and then set chils state*/
					break;

			}
		}
		va_end(list);
	}																													/* cleanup the system stack */
}

/* check for commands -> STATE_STOPPING means check for command stop... */
void checkCommands(brdkEM_typ* this, brdkEM_typ* parent, int numArgs, ...) {
	brdkEM_typ* child;
	int i,j;
	if(this->internal.cmdSC || this->cmd.abort || (this->cmd.stop && this->setup.skipStopSC)) {
		va_list list;																											/* define argument list variable */
		va_start(list, numArgs);																								/* init list */
		for(i=0; i < numArgs; i++) {
			switch(va_arg(list, brdk_em_states_typ)) {

				case STATE_STOPPING:
					if(this->cmd.stop) {
						i = numArgs;
						this->internal.pInterrupter = (unsigned long)this; /* module interrupted itself */
						this->state = STATE_STOPPING;
					}
					break;

				case STATE_RESETTING:
					if(this->cmd.reset) {
						i = numArgs;
						this->state = STATE_RESETTING;
					}
					break;

				case STATE_CLEARING:
					if(this->cmd.clear) {
						this->state = STATE_CLEARING;
					}
					break;

				case STATE_STARTING:
					if(this->cmd.start) {
						i = numArgs;
						this->state = STATE_STARTING;
					}
					break;

				case STATE_HOLDING:
					if(this->cmd.hold) {
						i = numArgs;
						this->internal.pInterrupter = (unsigned long)this; /* module interrupted itself */
						this->state = STATE_HOLDING;
					}
					break;

				case STATE_UNHOLDING:
					if(this->cmd.start) {
						i = numArgs;
						this->state = STATE_UNHOLDING;
					}
					break;

				case STATE_SUSPENDING:
					if(this->cmd.suspend) {
						i = numArgs;
						this->internal.pInterrupter = (unsigned long)this; /* module interrupted itself */
						this->state = STATE_SUSPENDING;
					}
					break;

				case STATE_UNSUSPENDING:
					if(this->cmd.start) {
						i = numArgs;
						this->state = STATE_UNSUSPENDING;
					}
					break;

				case STATE_COMPLETING:
					if(this->cmd.complete) {
						i = numArgs;
						this->state = STATE_COMPLETING;
					}
					break;

				case STATE_ABORTING:
					if(this->cmd.abort) {
						i = numArgs;
						this->internal.pInterrupter = (unsigned long)this; /* module interrupted itself */
						this->state = STATE_ABORTING;
					}
					break;

				case STATE_ACTIVATING:
					/* wait for initialization complete */
					if(this->internal.initSubstate == 65000) {
						switch(this->setup.activation) {

							case BRDK_EM_ACTIVATE:
								this->state = STATE_ACTIVATING;
								break;

							case BRDK_EM_ACTIVATE_BY_PARENT:
								if(parent != NULL) {
									switch(parent->state) {
										case STATE_DEACTIVATING: case STATE_DEACTIVATED: setSubStateText(this,(unsigned long)"waiting for parent's activation"); break;
										default:
											if(!parent->internal.deactivateRequest) this->state = STATE_ACTIVATING;
											break;
									}
								}
								break;

							default:
								setSubStateText(this, (unsigned long)"waiting for activation");
								break;

						}
					}
					break;

				case STATE_DEACTIVATING:
					switch(this->setup.activation) {

						case BRDK_EM_DEACTIVATE:
							this->internal.deactivateRequest = true;
							for(j=0; j <= BRDK_EM_MAX_CHILDREN; j++) {		/* check all children */
								child = getEm(this->internal.muList.childrenIdx[j]);
								if(child != NULL) {
									if(child->state != STATE_DEACTIVATED && child->state && STATE_DEACTIVATING) break;
								}
							}
							if(j > BRDK_EM_MAX_CHILDREN) {
								i = numArgs;
								this->state = STATE_DEACTIVATING;
							}
							break;

						case BRDK_EM_ACTIVATE_BY_PARENT:
							if(parent != NULL) {
								switch(parent->state) {
									case STATE_DEACTIVATING: case STATE_DEACTIVATED: this->state = STATE_DEACTIVATING; break;

									case STATE_ABORTED: case STATE_STOPPED:
										/* check if parent has deactivation command and then follow */
										if(parent->internal.deactivateRequest) {
											this->internal.deactivateRequest = true;
											for(j=0; j <= BRDK_EM_MAX_CHILDREN; j++) {		/* check all children */
												child = getEm(this->internal.muList.childrenIdx[j]);
												if(child != NULL) {
													if(child->state != STATE_DEACTIVATED && child->state && STATE_DEACTIVATING) break;
												}
											}
											if(j > BRDK_EM_MAX_CHILDREN) {
												i = numArgs;
												this->state = STATE_DEACTIVATING;
											}
										}
										break;

									default: break;
								}
							}
							break;

						default:
							break;

					}
					break;

				default:
					break;

			}
		}
		va_end(list);
		/* check if an unvalid command has been given */
		this->status.unvalidatedCmd = this->state != this->internal.old.state ? false : this->cmd.abort || this->cmd.clear || this->cmd.stop || this->cmd.reset || this->cmd.start || this->cmd.hold || this->cmd.suspend || this->cmd.complete;
	}
}

/* Add's a child to the parents child list */
unsigned short RegisterChild(brdkEM_typ* this, brdkEM_typ* parent) {
	int i=0, j=0;
	if(parent != NULL) {
		for(i=0; i < BRDK_EM_MAX_CHILDREN; i++) {
			if(parent->internal.muList.childrenIdx[i] == this->internal.muList.idx) break;	/* child already exists in array. index is returned */
			else if(parent->internal.muList.childrenIdx[i] == -1) {							/* finds an empty spot in the array */
				j = SemAcquire(parent->internal.SemCreate_0.ident);							/* checks if the semaphore is free */
				if(j == ERR_OK) {
					parent->internal.muList.childrenIdx[i] = this->internal.muList.idx;		/* puts the index in the array */
					parent->status.childCount++;
					SemRelease(parent->internal.SemCreate_0.ident);							/* releases the semaphore again */
					i = ERR_OK;
				}
				else {
					i = j;	/* 33322: Semaphore with the specified ident does not exist   33323: Semaphore is being used */
					if(this->setup.status.stateSubstateMode) {
						brdkStrCpy((unsigned long)tmpStr,(unsigned long)"semaphore error: ");
						brdkStrAppendUdintToA(j,(unsigned long)tmpStr,10,-1);
						setSubStateText(this,(unsigned long)tmpStr);
					}
				}
				break;
			}
		}
		if(i == BRDK_EM_MAX_CHILDREN) {  /* error: child array too small. Solution: make child array bigger */
			setSubStateText(this,(unsigned long)"parent child array full. Increase BRDK_EM_MAX_CHILDREN.");
		}
	}
	return i;
}

/* Unregister a child */
unsigned short UnregisterChild(brdkEM_typ* this, brdkEM_typ* parent) {
	int i=65000,j;
	if(parent != NULL) {
		for(i=0; i < BRDK_EM_MAX_CHILDREN; i++) {
			if(parent->internal.muList.childrenIdx[i] == this->internal.muList.idx) {	/* child found */
				j = SemAcquire(parent->internal.SemCreate_0.ident);	/* checks if the semaphore is free */
				if(j == ERR_OK) {
					parent->internal.muList.childrenIdx[i] = -1;			/* pointer is removed from the array */
					parent->status.childCount--;
					for(j=i; j < BRDK_EM_MAX_CHILDREN; j++) parent->internal.muList.childrenIdx[j] = parent->internal.muList.childrenIdx[j+1];
					SemRelease(parent->internal.SemCreate_0.ident);		/* releases the semaphore again */
					i = ERR_OK;
					this->internal.muList.parentIdx = -1;
				}
				else {
					i = j;	/* 33322: Semaphore with the specified ident does not exist   33323: Semaphore is being used */
					if(this->setup.status.stateSubstateMode) {
						brdkStrCpy((unsigned long)tmpStr,(unsigned long)"semaphore error: ");
						brdkStrAppendUdintToA(j,(unsigned long)tmpStr,10,-1);
						setSubStateText(this,(unsigned long)tmpStr);
					}
				}
				break;
			}
		}
		if(i == BRDK_EM_MAX_CHILDREN) {  /* error: child not found in array */
			setSubStateText(this,(unsigned long)"child not found in parent array.");
		}
	}
	return i;
}
```

#### brdkEMSleep.c
```c
#include <brdkMU_func.h>

signed long brdkEMSleep(unsigned long pEM) {
	brdkEM_typ* this;
	if(pEM != 0) {
		this = (brdkEM_typ*)pEM;
		this->status.sleeping = true;
		if(this->setup.status.last) {
			brdkStrMemMove((unsigned long)this->status.last[1],(unsigned long)this->status.last[0], sizeof(this->status.last[0])*BRDK_MU_MAX_LAST_SIZE);
			brdkStrCpy((unsigned long)this->status.last[0],(unsigned long)"module put to sleep");
		}
		return sleepMU(this->internal.muList.idx, pEM);
	}
	return -1;
}
```

### Program Logical/Modules/Main/Main (IEC)

#### Variables.var
```iecst
VAR
	em : brdkEM;
	MC_BR_MoveInPlane_Acp6D_0 : MC_BR_MoveInPlane_Acp6D;
	modeSelectorOldValue : driveModes;
	TON_0 : TON;
	MC_BR_AsmReboot_Acp6D_0 : MC_BR_AsmReboot_Acp6D;
	MC_BR_AsmHalt_Acp6D_0 : MC_BR_AsmHalt_Acp6D;
END_VAR
```

### Types.typ
```iecst
TYPE
	gMain_par_typ : 	STRUCT
		itemsPrShuttle : INT;
		controlLight : BOOL;
	END_STRUCT;
	gMain_status_typ : 	STRUCT
		powerOff : INT;
		running : INT;
		powerOn : INT;
		itemsPrHour : INT;
		itemsPrMin : INT;
		error : INT;
	END_STRUCT;
	gMain_cmd_typ : 	STRUCT
		powerOff : BOOL;
		powerOn : BOOL;
		start : BOOL;
		pause : BOOL;
		reset : BOOL;
		stop : BOOL;
		restartCtrl : BOOL; (*WARNING: restarts 6D controller and PLC*)
	END_STRUCT;
	gMain_typ : 	STRUCT
		par : gMain_par_typ;
		status : gMain_status_typ;
		cmd : gMain_cmd_typ;
	END_STRUCT;
END_TYPE
```

### Program Logical/Modules/Acopos6D/Acopos6D (IEC)

#### Main.st - Init, cyclic, exit code
```iecst
PROGRAM _INIT
	em.setup.name := 'Acopos6D';
	em.setup.parent.name := 'main';
	em();

	MC_BR_AsmGetInfo_Acp6D_0.Assembly			:= ADR(gAssembly6D_1);
	MC_BR_AsmGetShuttle_Acp6D_0.Assembly 		:= ADR(gAssembly6D_1);
	MC_BR_AsmReadStatus_Acp6D_0.Assembly 		:= ADR(gAssembly6D_1);
	MC_BR_AsmPowerOn_Acp6D_0.Assembly			:= ADR(gAssembly6D_1);
	MC_BR_AsmPowerOff_Acp6D_0.Assembly			:= ADR(gAssembly6D_1);
	MC_BR_AsmStop_Acp6D_0.Assembly				:= ADR(gAssembly6D_1);
	MC_BR_MoveInPlaneAsync_Acp6D_0.Assembly		:= ADR(gAssembly6D_1);
	MC_BR_ShGroupCreate_Acp6D_0.Assembly 		:= ADR(gAssembly6D_1);
	MC_BR_ShGroupCreate_Acp6D_1.Assembly 		:= ADR(gAssembly6D_1);
	MC_BR_ShGroupCreate_Acp6D_2.Assembly 		:= ADR(gAssembly6D_1);
	MC_BR_ShGroupCreate_Acp6D_3.Assembly 		:= ADR(gAssembly6D_1);
	MC_BR_ShGroupCreate_Acp6D_4.Assembly		:= ADR(gAssembly6D_1);
	MC_BR_MacroCreate_Acp6D_0.Assembly			:= ADR(gAssembly6D_1);
	MC_BR_AsmLevitation_Acp6D_0.Assembly		:= ADR(gAssembly6D_1);

	MC_BR_AsmReadStatus_Acp6D_0.Enable			:= TRUE;
	//MC_BR_AsmGetInfo_Acp6D_0.Execute := TRUE;

	MC_BR_AsmReadStatus_Acp6D_0();
END_PROGRAM

PROGRAM _CYCLIC
	// Setup config parameters
	config;

	// IF 6D Controller goes into Error PackML State machine will follow
	IF MC_BR_AsmReadStatus_Acp6D_0.Valid AND MC_BR_AsmReadStatus_Acp6D_0.AssemblyErrorStop THEN
		em.cmd.abort := TRUE;
	END_IF

	CASE em.state OF
		STATE_STOPPED:
			em.description := 'Waiting for reset cmd';
			IF MC_BR_AsmReadStatus_Acp6D_0.AssemblyDisabled AND NOT MC_BR_AsmReadStatus_Acp6D_0.AssemblyErrorStop THEN
				em.cmd.sc := TRUE;
			ELSE
				em.cmd.sc := FALSE;
			END_IF

		STATE_RESETTING:
			CASE em.substate OF
				0:
					em.description := 'Reset all inputs';
					ResetInput;
					em.substate := 2;

				2:
					MC_BR_AsmGetInfo_Acp6D_0.Execute := TRUE;
					IF MC_BR_AsmGetInfo_Acp6D_0.Done THEN
						gAcp6DCtrl.Status.currentNumShuttles := MC_BR_AsmGetInfo_Acp6D_0.AssemblyInfo.NumberOfShuttles;
						localCurrentNumShuttles := gAcp6DCtrl.Status.currentNumShuttles;
						MC_BR_AsmGetInfo_Acp6D_0.Execute := FALSE;
						IF gAcp6DCtrl.Status.currentNumShuttles > 0 THEN
							em.substate := 5;
						ELSE
							em.cmd.abort := TRUE;
						END_IF
					END_IF

				5:
					em.description := 'Load shuttle IDs';
					MC_BR_AsmGetShuttle_Acp6D_0.Enable := TRUE;
					gAcp6DCtrl.Status.currentNumShuttles := MC_BR_AsmGetInfo_Acp6D_0.AssemblyInfo.NumberOfShuttles;
					IF MC_BR_AsmGetShuttle_Acp6D_0.Valid AND MC_BR_AsmGetShuttle_Acp6D_0.Busy THEN
						tempCounter := 0;
						em.substate := 6;
					END_IF

				6:
					em.description := 'copy shuttle ref';
					MC_BR_AsmGetShuttle_Acp6D_0.Next := FALSE;
					gAcp6DCtrl.Status.ShuttleInfo[MC_BR_AsmGetShuttle_Acp6D_0.AdditionalInfo.ShuttleID-1].ID := MC_BR_AsmGetShuttle_Acp6D_0.AdditionalInfo.ShuttleID;
					gAcp6DCtrl.Status.ShuttleInfo[MC_BR_AsmGetShuttle_Acp6D_0.AdditionalInfo.ShuttleID-1].shuttleRef := MC_BR_AsmGetShuttle_Acp6D_0.Shuttle;
					IF MC_BR_AsmGetShuttle_Acp6D_0.RemainingCount = 0 THEN
						//MC_BR_AsmGetShuttle_Acp6D_0.Enable := FALSE;
						em.substate := 10;
					ELSE
						em.substate := 7;
					END_IF

				7:
					MC_BR_AsmGetShuttle_Acp6D_0.Next := TRUE;
					em.substate := 6;

				10:
					em.description := 'Power on 6DController';
					IF MC_BR_AsmReadStatus_Acp6D_0.AssemblyReady THEN
						em.substate := 15;
					ELSE
						MC_BR_AsmPowerOn_Acp6D_0.Execute 			:= TRUE;
						IF(MC_BR_AsmPowerOn_Acp6D_0.Acknowledge AND MC_BR_AsmPowerOn_Acp6D_0.Done)THEN
							MC_BR_AsmPowerOn_Acp6D_0.Execute 		:= FALSE;
							em.substate  							:= 15;
						ELSIF(MC_BR_AsmPowerOn_Acp6D_0.Error)THEN
							MC_BR_AsmPowerOn_Acp6D_0.Execute 		:= FALSE;
							em.cmd.abort							:= TRUE;
						END_IF;
					END_IF

				15:
					em.description := 'Check Assembly Ready';
					IF MC_BR_AsmReadStatus_Acp6D_0.AssemblyReady THEN
						em.substate := 23;
						tempShuttleCnt := 0;
					ELSE
						em.substate := 10; //Sometimes AsmPowerOn dont power on the system
					END_IF

				23:
					em.description := 'Break all shuttles';
					MC_BR_AsmStop_Acp6D_0.Execute := TRUE;
					IF MC_BR_AsmStop_Acp6D_0.Done THEN
						MC_BR_AsmStop_Acp6D_0.Execute := FALSE;
						em.substate := 25;
					END_IF

				25:
					em.description := 'Check all shuttles states';
					IF gAcp6DCtrl.Status.ShuttleInfo[tempShuttleCnt].State = mcACP6D_SH_STATE_IDLING THEN
						tempShuttleCnt := tempShuttleCnt + 1;
						em.substate := 27;
					ELSE
						em.substate := 15;
					END_IF

				27:
					em.description := 'all shuttles checked?';
					IF tempShuttleCnt > localCurrentNumShuttles-1 THEN
						em.substate := 40;
					ELSE
						em.substate := 25;
					END_IF

				40:
					em.description := 'Check one shuttle to see if MoveInPlaceAsync is done';
					IF gAcp6DCtrl.Status.ShuttleInfo[0].State =  mcACP6D_SH_STATE_IDLING THEN
						em.substate := 90; //cant use Async when stereoType is defined
					END_IF

				90:
					shuttleGroups;
					macroCreatorAction;
					IF createShGroup = 100 AND macroCreater = 70 THEN
						em.substate := 100;
					END_IF

				100:
					MC_BR_ShGroupGetInfo_Acp6D_0.ShuttleGroup := shGroupShuttle1_2;
					MC_BR_ShGroupGetInfo_Acp6D_0.Execute := TRUE;
					em.cmd.sc := TRUE;
			END_CASE

		STATE_STARTING:
			CASE em.substate OF
				0:
					FOR i := 0 TO NUM_SHUTTLES DO
						IF gAcp6DCtrl.Status.ShuttleInfo[i].State = mcACP6D_SH_STATE_IDLING OR gAcp6DCtrl.Status.ShuttleInfo[i].State = mcACP6D_SH_STATE_LANDED THEN
						ELSE
							EXIT;
						END_IF
					END_FOR
					IF i > NUM_SHUTTLES THEN
						em.substate := 2;
					END_IF

				2:
					em.description := 'Break all shuttles';
					MC_BR_AsmStop_Acp6D_0.Execute := TRUE;
					IF MC_BR_AsmStop_Acp6D_0.Done THEN
						MC_BR_AsmStop_Acp6D_0.Execute := FALSE;
						em.substate := 3;
					END_IF

				3:
					FOR i := 0 TO NUM_SHUTTLES DO
						IF gAcp6DCtrl.Status.ShuttleInfo[i].State = mcACP6D_SH_STATE_IDLING OR gAcp6DCtrl.Status.ShuttleInfo[i].State = mcACP6D_SH_STATE_LANDED THEN
						ELSE
							EXIT;
						END_IF
					END_FOR
					IF i > NUM_SHUTTLES THEN
						em.substate := 5;
					END_IF

				5:
					em.description := 'Move to start pos';
					TON_watchdog.IN := FALSE; // Firmware bugfix
					TON_watchdog.PT := t#4s; // Firmware bugfix
					MC_BR_MoveInPlaneAsync_Acp6D_0.Parameters.Acceleration := gAcp6DCtrl.Par.Acceleration;
					MC_BR_MoveInPlaneAsync_Acp6D_0.Parameters.Velocity := gAcp6DCtrl.Par.Velocity;
					FOR i := 0 TO UINT_TO_USINT(localCurrentNumShuttles-1) DO
						MC_BR_MoveInPlaneAsync_Acp6D_0.Parameters.AsyncPar[i].Shuttle := ADR(gAcp6DCtrl.Status.ShuttleInfo[i].shuttleRef);
						MC_BR_MoveInPlaneAsync_Acp6D_0.Parameters.AsyncPar[i].X := shuttleStartupInfo[i].initXPos;
						MC_BR_MoveInPlaneAsync_Acp6D_0.Parameters.AsyncPar[i].Y := shuttleStartupInfo[i].initYPos;
					END_FOR
					MC_BR_MoveInPlaneAsync_Acp6D_0.Execute := TRUE;
					IF MC_BR_MoveInPlaneAsync_Acp6D_0.Done THEN
						MC_BR_MoveInPlaneAsync_Acp6D_0.Execute := FALSE;
						em.substate := 10;
					END_IF
					// Firmware bugfix - Sometimes MoveInPlaneAsync is stuck and will need a FB reset
//					IF MC_BR_MoveInPlaneAsync_Acp6D_0.Busy THEN
//						TON_watchdog.IN := TRUE;
//						IF TON_watchdog.Q THEN
//							MC_BR_MoveInPlaneAsync_Acp6D_0.Execute := FALSE;
//						END_IF
//					END_IF

				10:
					em.cmd.sc := TRUE;
			END_CASE

		STATE_EXECUTE:
			em.description := 'Shuttle program with selected mode is running';
			gAcp6DCtrl.Status.Ready := TRUE;
			em.cmd.sc := TRUE;

			CASE em.substate OF
				0:
					CASE gAcp6DCtrl.Par.modeSelector OF
						weight: em.substate := 2000;
						linkMovement: em.substate := 3000;
						dialGauge: em.substate := 7000;
						workstationMovement: em.substate := 8000;
						conveyorStationMovement: em.substate := 9000;
						flaskProgram: em.substate := 12000;
						boxProgram: em.substate := 13000;
						rotationProgram: em.substate := 14000;
						steelSheet: em.substate := 15000;
						test: em.substate := 16000;
						smartLab: em.substate := 17000;

					END_CASE

				2000..2999:
					enableButtons := FALSE;
					em.cmd.sc := FALSE;
					em.description := 'Weight Program';
					IF controlLight.weightProgram THEN
						lightValue := 12;
					END_IF

					FOR i := 0 TO NUM_SHUTTLES DO
						pShuttle ACCESS ADR(gShuttles[i]);
						cm ACCESS ADR (gShuttles[i].cm);
						pShuttle.cm.setup.parent.name := 'main';
						pShuttle.cm.setup.nameIdx := i;
						pShuttle.par.shuttleID := i;

						//Chosen action pr shuttle
						CASE i OF
							0:weightProgram;
							3:MovementRx;
							2:MovementRy;
							1:MovementZ;
						END_CASE
					END_FOR
					em.cmd.sc := TRUE;

				3000..3999:
						em.description := 'linkMovement Program';
						IF controlLight.linkProgram THEN
							lightValue := 1;
						END_IF

						linkMovementProgram;

				7000:
					em.description := 'dialGauge Program';
					IF controlLight.shuttlePrecision THEN
						lightValue := 3;
					END_IF

					FOR i := 0 TO NUM_SHUTTLES DO
						pShuttle ACCESS ADR(gShuttles[i]);
						cm ACCESS ADR (gShuttles[i].cm);
						pShuttle.cm.setup.parent.name := 'main';
						pShuttle.cm.setup.nameIdx := i;
						pShuttle.par.shuttleID := i;

						//Chosen action pr shuttle
						CASE i OF
							6: BasicMoveDialGauge;
							1: MovementZ;
							2: MovementRx;
							3: MovementRy;
						END_CASE
					END_FOR
					em.cmd.sc := TRUE;

				8000..8005:
					workStationSetup;

				8006..8999:
					workStationSetup;
					em.description := 'intelligentMovement';
					IF controlLight.intelligentMovementProgram THEN
						lightValue := 4;
					END_IF
						FOR i := 0 TO NR_OF_WORKSTATIONS DO
							pWorkstation ACCESS ADR (gWorkstations[i]);
							cm ACCESS ADR (gWorkstations[i].cm);
							pWorkstation.cm.setup.parent.name := 'main';
							//pShuttle.cm.setup.nameIdx := i;
							workStationMovement;
						END_FOR

				9000..9005:
					IF controlLight.intelligentMovementProgram THEN
						lightValue := 2;
					END_IF
					conveyorStationSetup;

				9006..9999:
					em.description := 'ConveyorMovement';

					conveyorStationSetup;
					FOR i := 0 TO NR_OF_WORKSTATIONS DO
						pWorkstation ACCESS ADR (gWorkstations[i]);
						cm ACCESS ADR (gWorkstations[i].cm);
						pWorkstation.cm.setup.parent.name := 'main';
						//pShuttle.cm.setup.nameIdx := i;
						conveyourStationMovement;
					END_FOR

				12000..12019:
					em.description := 'Flask Program';
					lightValue := 5;
					flaskProgramTask;

				12020..12999:
						em.description := 'Flask Program';
						flaskProgramTask;
						FOR i := 0 TO NUM_SHUTTLES-1 DO
							pShuttle ACCESS ADR(gShuttles[i]);
							cm ACCESS ADR (gShuttles[i].cm);
							pShuttle.cm.setup.parent.name := 'main';
							pShuttle.cm.setup.nameIdx := i;
							pShuttle.par.shuttleID := i;

							//Chosen action pr shuttle
							CASE i OF
								0:MovementRy;
								1:MovementZ;
								2:MovementRx;
							END_CASE
						END_FOR

				13000..13999:
					em.description := 'Box Program';
					lightValue := 7;
					boxProgramTask;

				14000..14049:
					em.description := 'Rotation program';
					lightValue := 9;
					em.cmd.sc := FALSE;
					rotationTask;

				14050..14999:
					em.description := 'Rotation program';
					em.cmd.sc := FALSE;
					FOR i := 0 TO NR_OF_WORKSTATIONS DO
						pWorkstation ACCESS ADR (gWorkstations[i]);
						cm ACCESS ADR (gWorkstations[i].cm);
						pWorkstation.cm.setup.parent.name := 'main';
						rotationStation;
					END_FOR
					rotationTask; // Controls em.cmd.sc so the program can be stopped at the correct time.

				15000..15009:
					em.description := 'Steelsheet program';
					lightValue := 6;
					steelSheetTask;

				15010..15999:
					em.description := 'Steelsheet program';
					FOR i := 0 TO NR_OF_WORKSTATIONS DO
						pWorkstation ACCESS ADR (gWorkstations[i]);
						cm ACCESS ADR (gWorkstations[i].cm);
						pWorkstation.cm.setup.parent.name := 'main';
						steelSheetStation;
					END_FOR

				16000..16009:
					em.description := 'Test program - Setup';
					testProgram;

				16010..16999:
					em.description := 'Test program - Movements';
					testProgram;
					FOR i := 0 TO NUM_SHUTTLES DO
						cm ACCESS ADR (gShuttles[i].cm);
						pShuttle ACCESS ADR(gShuttles[i]);
						pShuttle.cm.setup.parent.name := 'main';
						pShuttle.cm.setup.nameIdx := i;
						pShuttle.par.shuttleID := i;

						CASE i OF
							0..3: testMovements;
						END_CASE
					END_FOR

				17000..17009:
					em.description := 'Smart Lab program - Setup';
					smartLabSetup;

				17010..17014:

					em.description := 'Smart Lab Program - Write order if it has been placed';

					// The user has requested an order which is added to the buffer
					IF executeOrder THEN

						TON_0.PT := REAL_TO_TIME(200);
						TON_0.IN := TRUE;
						IF TON_0.Q THEN
							TON_0.IN := FALSE;
							executeOrder := FALSE;

							// If the buffer is empty go to read state, else just continue executing the order
//							IF bufferEmpty THEN
//								em.substate := 17015;
//							ELSE
//								em.substate := 17020;
//							END_IF

							// Write the order if the buffer is not full
							IF NOT bufferFull THEN
								writeOrder;
							END_IF

							em.substate := 17015;
						END_IF
					END_IF

				17015..17019:
					em.description := 'Smart Lab Program - Read order if the shuttles are ready to';

					// Read a new order if the entire other order has been initiated and the buffer is not empty
					IF remainingOrderAmount = 0 AND NOT bufferEmpty THEN
						// Read the order
						readOrder;

						// Create the route sheet
						CreateRouteSheet_0.inputProductOrder := productOrder;
						CreateRouteSheet_0();

						remainingOrderAmount := productOrder.amount;
						activeShuttles := activeShuttles + productOrder.amount;
						amountProductsFinished := 0;
					END_IF

					em.substate := 17020;

				17020..17999:
					em.description := 'Smart Lab program - Workstation movement';
					// Go through the workstations and run program for these
					FOR i := 0 TO (smartLabNumWorkstations - 1) DO
						pWorkstation ACCESS ADR (gWorkstations[i]);
						cm ACCESS ADR (gWorkstations[i].cm);
						pWorkstation.cm.setup.parent.name := 'main';
						pWorkstation.par.workstationID := i;

						smartLabWorkstationOperation;
					END_FOR

					// Go through the shuttles and run program for these
					FOR i := 0 TO (smartLabNumShuttles - 1) DO
						pShuttle ACCESS ADR(gShuttles[i]);
						cm ACCESS ADR (gShuttles[i].cm);
						pShuttle.cm.setup.parent.name := 'main';
						pShuttle.par.shuttleID := i;

						pShuttlePlan ACCESS ADR(shuttlePlans[pShuttle.par.shuttleID]);

						smartLabShuttleMovement;
					END_FOR

					// Go to write order if a new order is made or there are no active orders
					IF executeOrder THEN
						em.substate := 17010;
					END_IF

			END_CASE

		STATE_STOPPING,STATE_ABORTING:
			ResetInput;
			em.description := 'Power off 6D System';
			CASE em.substate OF
				0:
					IF MC_BR_AsmReadStatus_Acp6D_0.AssemblyReady OR MC_BR_AsmReadStatus_Acp6D_0.AssemblyHoming THEN
						em.substate := 10;
					ELSE
						em.substate := 100;
					END_IF

				10:
					em.description := 'Break all shuttles and shut down the system';
					MC_BR_AsmPowerOff_Acp6D_0.Execute := TRUE;
					IF MC_BR_AsmPowerOff_Acp6D_0.Done THEN
						ResetInput; //Reset all FB
						createShGroup := 0;
						MC_BR_AsmPowerOff_Acp6D_0.Execute := FALSE;
						em.substate := 100;
					END_IF

				100:
					em.description := 'Check if system is off';
					createShGroup := 0;
					em.cmd.sc := TRUE;
			END_CASE

		STATE_COMPLETING:
			ResetInput;
			em.description := 'Break all shuttles and clear Motion Buffer';
			CASE em.substate OF
				0:
					em.description := 'Break all shuttles';
					MC_BR_AsmStop_Acp6D_0.Execute := TRUE;
					IF MC_BR_AsmStop_Acp6D_0.Done THEN
						MC_BR_AsmStop_Acp6D_0.Execute := FALSE;
						tempCounter := 0;
						em.substate := 5;
					END_IF

				5:
					FOR i := 0 TO NUM_SHUTTLES DO
						IF gAcp6DCtrl.Status.ShuttleInfo[i].State = mcACP6D_SH_STATE_IDLING OR gAcp6DCtrl.Status.ShuttleInfo[i].State = mcACP6D_SH_STATE_LANDED THEN
						ELSE
							EXIT;
						END_IF
					END_FOR
					IF i > NUM_SHUTTLES THEN
						em.substate := 10;
					END_IF

				10:
					em.description := 'Levitate if any shuttle is landed';
					MC_BR_AsmLevitation_Acp6D_0.Parameters.Speed := 5; //1-5
					MC_BR_AsmLevitation_Acp6D_0.Parameters.Level := 1;
					MC_BR_AsmLevitation_Acp6D_0.Execute := TRUE;
					IF MC_BR_AsmLevitation_Acp6D_0.Done THEN
						MC_BR_AsmLevitation_Acp6D_0.Execute := FALSE;
						em.substate := 100;
					END_IF
					IF MC_BR_AsmLevitation_Acp6D_0.Error THEN
						em.cmd.abort := TRUE;
					END_IF

				100:
					FOR i := 0 TO NUM_SHUTTLES DO
						IF gAcp6DCtrl.Status.ShuttleInfo[i].State = mcACP6D_SH_STATE_IDLING THEN
						ELSE
							EXIT;
						END_IF
					END_FOR
					IF i > NUM_SHUTTLES THEN
						em.substate := 110;
					END_IF

				110:
					ResetInput;
					em.cmd.reset := TRUE;
					em.cmd.sc := TRUE;
			END_CASE

		ELSE
			em.cmd.sc := TRUE;
	END_CASE

	//Shuttle pos update
	FOR i := 0 TO NUM_SHUTTLES DO
		// check there is a shuttle
		IF gAcp6DCtrl.Status.ShuttleInfo[i].shuttleRef.controlif > 0 THEN
			MC_BR_ShReadInfo_Acp6D_0[i].Shuttle := ADR(gAcp6DCtrl.Status.ShuttleInfo[i].shuttleRef);
			MC_BR_ShReadInfo_Acp6D_0[i].Enable := TRUE;
			gAcp6DCtrl.Status.ShuttleInfo[i].Position := MC_BR_ShReadInfo_Acp6D_0[i].ShuttleInfo.Position;
			gAcp6DCtrl.Status.ShuttleInfo[i].State := MC_BR_ShReadInfo_Acp6D_0[i].ShuttleInfo.State;
			MC_BR_ShReadInfo_Acp6D_0[i]();

			//Turn off system if shuttle is not detected (removed by hand)
			IF em.state = STATE_EXECUTE AND (MC_BR_ShReadInfo_Acp6D_0[i].ShuttleInfo.State = mcACP6D_SH_STATE_RESERVED OR MC_BR_ShReadInfo_Acp6D_0[i].ShuttleInfo.State = mcACP6D_SH_STATE_DISABLED) THEN
				em.cmd.abort := TRUE;
			END_IF
		END_IF
	END_FOR

	em();
	MC_BR_AsmGetShuttle_Acp6D_0();
	MC_BR_AsmReadStatus_Acp6D_0();
	MC_BR_AsmPowerOn_Acp6D_0();
	MC_BR_AsmPowerOff_Acp6D_0();
	MC_BR_AsmStop_Acp6D_0();
	MC_BR_AsmLevitation_Acp6D_0();
	MC_BR_MoveInPlaneAsync_Acp6D_0();
	MC_BR_ShLevitation_Acp6D_0();
	MC_BR_MoveInPlane_Acp6D_0();
	MC_BR_MoveArc_Acp6D_0();
	MC_BR_ShGroupCreate_Acp6D_0();
	MC_BR_ShGroupCreate_Acp6D_1();
	MC_BR_ShGroupCreate_Acp6D_2();
	MC_BR_ShGroupCreate_Acp6D_3();
	MC_BR_ShGroupCreate_Acp6D_4();
	MC_BR_ShGroupAddShuttle_Acp6D_0();
	MC_BR_ShGroupCoupleCtrl_Acp6D_0();
	MC_BR_ShGroupGetInfo_Acp6D_0();
	MC_BR_ReadCyclicPosition_Acp6D_0();
	MC_BR_ReadCyclicPosition_Acp6D_1();
	MC_BR_ReadCyclicPosition_Acp6D_2();
	MC_BR_ReadCyclicPosition_Acp6D_3();
	MC_BR_MacroCreate_Acp6D_0();
	MC_BR_Move6D_Acp6D_0();
	MC_BR_MacroRun_Acp6D_0();
	MC_BR_MacroSave_Acp6D_0();
	MC_BR_AsmGetInfo_Acp6D_0();
	MC_BR_RotaryMotionSpin_Acp6D_0();
	MC_BR_RotaryMotion_Acp6D_0();
	TON_watchdog();
	TON_0();

END_PROGRAM

PROGRAM _EXIT
	(* Insert code here *)

END_PROGRAM
```

#### Config.st
```iecst
ACTION config:
	gAcp6DCtrl.Status.Ready := FALSE;
	gameBrain.showHMIButton := FALSE;
	enableButtons := TRUE;

	shuttleStartupInfo[0].initXPos := 0.060;
	shuttleStartupInfo[0].initYPos := 0.060;
	shuttleStartupInfo[1].initXPos := 0.180;
	shuttleStartupInfo[1].initYPos := 0.180;
	shuttleStartupInfo[2].initXPos := 0.300;
	shuttleStartupInfo[2].initYPos := 0.060;
	shuttleStartupInfo[3].initXPos := 0.420;
	shuttleStartupInfo[3].initYPos := 0.180;

	shuttleStartupInfo[4].initXPos := 0.540;
	shuttleStartupInfo[4].initYPos := 0.060;
	shuttleStartupInfo[5].initXPos := 0.660;
	shuttleStartupInfo[5].initYPos := 0.180;
	shuttleStartupInfo[6].initXPos := 0.060;
	shuttleStartupInfo[6].initYPos := 0.300;
	shuttleStartupInfo[7].initXPos := 0.180;
	shuttleStartupInfo[7].initYPos := 0.420;

//	shuttleStartupInfo[8].initXPos := 0.300;
//	shuttleStartupInfo[8].initYPos := 0.300;
//	shuttleStartupInfo[9].initXPos := 0.420;
//	shuttleStartupInfo[9].initYPos := 0.420;

END_ACTION
```

#### ResetInput.st
```iecst
ACTION ResetInput:
	MC_BR_AsmPowerOff_Acp6D_0.Execute		:= FALSE;
	MC_BR_AsmPowerOn_Acp6D_0.Execute		:= FALSE;
	MC_BR_ReadCyclicPosition_Acp6D_0.Enable	:= FALSE;
	MC_BR_ReadCyclicPosition_Acp6D_1.Enable	:= FALSE;
	MC_BR_ReadCyclicPosition_Acp6D_2.Enable	:= FALSE;
	MC_BR_ReadCyclicPosition_Acp6D_3.Enable	:= FALSE;
	gAcp6DCtrl.Cmd.PowerOn					:= FALSE;
	gAcp6DCtrl.Cmd.PowerOff					:= FALSE;
	gAcp6DCtrl.Cmd.StartProcess				:= FALSE;
	gAcp6DCtrl.Cmd.StopProcess				:= FALSE;

	ABBRobot.returnBigWeightMovement 		:= FALSE;
	ABBRobot.returnSmallWeightMovement		:= FALSE;
	ABBRobot.startBigWeightMovement			:= FALSE;
	ABBRobot.startSmallWeightMovement		:= FALSE;

	MC_BR_MoveInPlane_Acp6D_0.Execute := FALSE;
	MC_BR_MoveInPlane_Acp6D_0.Parameters.Mode := 0;
	MC_BR_MoveInPlane_Acp6D_0.Parameters.Path := 0;

	FOR i := 0 TO NR_OF_WORKSTATIONS DO
		gWorkstations[i].cm.state := 0;
		gWorkstations[i].MC_BR_ShLevitation_Acp6D_0.Execute := FALSE;
		gWorkstations[i].MC_BR_MoveArc_Acp6D_0.Execute := FALSE;
		gWorkstations[i].MC_BR_MoveInPlane_Acp6D_0.Execute := FALSE;
		gWorkstations[i].MC_BR_RotaryMotion_Acp6D_0.Execute := FALSE;
		gWorkstations[i].MC_BR_RotaryMotionSpin_Acp6D_0.Execute := FALSE;
		gWorkstations[i].MC_BR_Move6D_Acp6D_0.Execute := FALSE;
		gWorkstations[i].par.ArcMovement := FALSE;
		gWorkstations[i].par.landBeforeProcess := FALSE;
		gWorkstations[i].par.pathRouting := FALSE;
		gWorkstations[i].par.processTime := FALSE;
		gWorkstations[i].par.tempShuttleID := FALSE;
		gWorkstations[i].par.xLocation := FALSE;
		gWorkstations[i].par.yLocation := FALSE;
		gWorkstations[i].TON_0.IN := FALSE;
		gWorkstations[i].par.xLocation										:= 0.0;
		gWorkstations[i].par.yLocation										:= 0.0;
		gWorkstations[i].par.nextStationSelector							:= '0';
		gWorkstations[i].par.processTime									:= 0;
		gWorkstations[i].par.pathRouting									:= 0;
		gWorkstations[i].par.ArcMovement									:= FALSE;
		gWorkstations[i].par.landBeforeProcess								:= FALSE;
	END_FOR

	FOR i := 0 TO NUM_SHUTTLES DO
		gShuttles[i].function.MC_BR_Move6D_Acp6D_0.Execute := FALSE;
		gShuttles[i].function.MC_BR_MoveInPlane_Acp6D_0.Execute := FALSE;
		gShuttles[i].function.MC_BR_MoveShortAxis_Acp6D_0.Execute := FALSE;
		gShuttles[i].function.TON_0.IN := FALSE;
		gShuttles[i].cm.state := 0;

		//MC_BR_ShReadInfo_Acp6D_0[i].Enable := FALSE;

		//MC_BR_MoveArc_Acp6D_0[i].Execute := FALSE;

		MC_BR_MoveShortAxis_Acp6D_0[i].Execute := FALSE;
	END_FOR

	FOR k := 0 TO 1 DO
		FOR j := 0 TO NUM_SHUTTLES DO
			//MC_BR_ReadCyclicChAxis_Acp6D_0[k,j].Enable := FALSE;
		END_FOR
	END_FOR

	TON_0.IN								:= FALSE;
	MC_BR_MoveArc_Acp6D_0.Execute 			:= FALSE;
	MC_BR_MoveInPlaneAsync_Acp6D_0.Execute	:= FALSE;
	MC_BR_MoveInPlane_Acp6D_0.Execute		:= FALSE;
	//MC_BR_ShReadInfo_Acp6D_0.Execute		:= FALSE;
	MC_BR_ShGroupCreate_Acp6D_0.Execute		:= FALSE;
	MC_BR_ShGroupAddShuttle_Acp6D_0.Execute := FALSE;
	MC_BR_ShGroupCoupleCtrl_Acp6D_0.Execute	:= FALSE;
	MC_BR_ShGroupGetInfo_Acp6D_0.Execute	:= FALSE;
	MC_BR_RotaryMotionSpin_Acp6D_0.Execute 	:= FALSE;
	MC_BR_AsmLevitation_Acp6D_0.Execute		:= FALSE;
	//MC_BR_MacroList_Acp6D_0.Execute			:= FALSE;
	//MC_BR_MacroLoad_Acp6D_0.Execute			:= FALSE;
	//MC_BR_MoveShortAxis_Acp6D_0.Execute		:= FALSE;
	//MC_BR_PlanetCtrl_Acp6D_0.Execute		:= FALSE;
	MC_BR_Move6D_Acp6D_0.Execute 			:= FALSE;
	MC_BR_ShLevitation_Acp6D_0.Execute	:= FALSE;

	//MC_BR_MacroList_Acp6D_0();
	//MC_BR_MacroLoad_Acp6D_0();

END_ACTION
```

#### BasicMovement.st
```iecst
ACTION BasicMoveDialGauge:
	pShuttle.function.MC_BR_MoveInPlane_Acp6D_0.Parameters.Acceleration := 5;
	pShuttle.function.MC_BR_MoveInPlane_Acp6D_0.Parameters.Velocity := 0.02;
	pShuttle.function.MC_BR_MoveInPlane_Acp6D_0.Shuttle := ADR(gAcp6DCtrl.Status.ShuttleInfo[pShuttle.par.shuttleID].shuttleRef);
	pShuttle.function.MC_BR_MoveInPlane_Acp6D_0.Parameters.Mode := 0; //Absolute
	pShuttle.function.MC_BR_MoveInPlane_Acp6D_0.Parameters.Path := 0; //direct

	CASE pShuttle.cm.state OF
		0:
			cm.description := 'Move shuttle to preDialPos';
			pShuttle.function.MC_BR_MoveInPlane_Acp6D_0.Parameters.Position.X := 0.060;
			pShuttle.function.MC_BR_MoveInPlane_Acp6D_0.Parameters.Position.Y := 0.300;
			pShuttle.function.MC_BR_MoveInPlane_Acp6D_0.Execute := TRUE;
			IF pShuttle.function.MC_BR_MoveInPlane_Acp6D_0.Acknowledge THEN
				pShuttle.function.MC_BR_MoveInPlane_Acp6D_0.Execute := FALSE;
				cm.state := 5;
			END_IF

		5:
			cm.description := 'Move shuttle to dialGauge';
			pShuttle.function.MC_BR_MoveInPlane_Acp6D_0.Parameters.Position.X := 0.050;
			pShuttle.function.MC_BR_MoveInPlane_Acp6D_0.Parameters.Position.Y := 0.300;
			pShuttle.function.MC_BR_MoveInPlane_Acp6D_0.Execute := TRUE;
			IF pShuttle.function.MC_BR_MoveInPlane_Acp6D_0.Acknowledge THEN
				pShuttle.function.MC_BR_MoveInPlane_Acp6D_0.Execute := FALSE;
				cm.state := 10;
			END_IF

		10:
			cm.description := 'Check pos reached';
			FOR i := 0 TO NUM_SHUTTLES DO
				IF((gAcp6DCtrl.Status.ShuttleInfo[pShuttle.par.shuttleID].Position.X > 0.050 - MARGIN AND gAcp6DCtrl.Status.ShuttleInfo[pShuttle.par.shuttleID].Position.X < 0.050 + MARGIN) AND
					gAcp6DCtrl.Status.ShuttleInfo[pShuttle.par.shuttleID].Position.Y > 0.300 - MARGIN AND gAcp6DCtrl.Status.ShuttleInfo[pShuttle.par.shuttleID].Position.Y < 0.300 + MARGIN) THEN
					IF gAcp6DCtrl.Status.ShuttleInfo[pShuttle.par.shuttleID].State = mcACP6D_SH_STATE_IDLING THEN
						cm.state := 20;
					END_IF
				END_IF
			END_FOR

		20:
			cm.description := 'Wait time';
			pShuttle.function.TON_0.PT := t#3s;
			pShuttle.function.TON_0.IN := TRUE;
			IF pShuttle.function.TON_0.Q THEN
				pShuttle.function.TON_0.IN := FALSE;
				cm.state := 30;
			END_IF

		30:
			cm.description := 'Move shuttle away from dialGauge';
			pShuttle.function.MC_BR_MoveInPlane_Acp6D_0.Parameters.Position.X := 0.060;
			pShuttle.function.MC_BR_MoveInPlane_Acp6D_0.Parameters.Position.Y := 0.300;
			pShuttle.function.MC_BR_MoveInPlane_Acp6D_0.Execute := TRUE;
			IF pShuttle.function.MC_BR_MoveInPlane_Acp6D_0.Acknowledge THEN
				pShuttle.function.MC_BR_MoveInPlane_Acp6D_0.Execute := FALSE;
				cm.state := 40;
			END_IF

		40:
			cm.description := 'Check pos reached';
			FOR i := 0 TO NUM_SHUTTLES DO
				IF((gAcp6DCtrl.Status.ShuttleInfo[pShuttle.par.shuttleID].Position.X > 0.060 - MARGIN AND gAcp6DCtrl.Status.ShuttleInfo[pShuttle.par.shuttleID].Position.X < 0.060 + MARGIN) AND
					gAcp6DCtrl.Status.ShuttleInfo[pShuttle.par.shuttleID].Position.Y > 0.300 - MARGIN AND gAcp6DCtrl.Status.ShuttleInfo[pShuttle.par.shuttleID].Position.Y < 0.300 + MARGIN) THEN
					IF gAcp6DCtrl.Status.ShuttleInfo[pShuttle.par.shuttleID].State = mcACP6D_SH_STATE_IDLING THEN
						cm.state := 0;
					END_IF
				END_IF
			END_FOR

	END_CASE

	cm();
	pShuttle.function.TON_0();
	pShuttle.function.MC_BR_MoveInPlane_Acp6D_0();

END_ACTION
```
